C01778=1011.519,353.301,-157.245,170.736,52.593,160.409
C01779=1011.528,353.615,-157.291,170.746,52.587,160.410
C01780=1011.537,353.929,-157.337,170.758,52.582,160.411
C01781=1011.545,354.243,-157.384,170.769,52.577,160.412
C01782=1011.554,354.557,-157.431,170.779,52.571,160.412
C01783=1011.562,354.804,-157.467,170.788,52.567,160.413
C01784=1011.569,355.052,-157.505,170.796,52.563,160.414
C01785=1011.576,355.299,-157.541,170.806,52.558,160.414
C01786=1011.582,355.546,-157.578,170.814,52.554,160.415
C01787=1011.590,355.793,-157.615,170.823,52.550,160.416
C01788=1011.597,356.041,-157.652,170.831,52.546,160.416
C01789=1011.604,356.287,-157.689,170.840,52.541,160.417
C01790=1011.612,356.534,-157.726,170.849,52.537,160.418
C01791=1011.619,356.782,-157.762,170.859,52.533,160.419
C01792=1011.626,357.029,-157.800,170.867,52.529,160.420
C01793=1011.633,357.276,-157.836,170.876,52.525,160.420
C01794=1011.641,357.523,-157.873,170.884,52.521,160.421
C01795=1011.648,357.770,-157.911,170.893,52.517,160.422
C01796=1011.655,358.018,-157.948,170.903,52.513,160.423
C01797=1011.662,358.265,-157.985,170.911,52.509,160.423
C01798=1011.669,358.512,-158.023,170.920,52.505,160.424
C01799=1011.676,358.759,-158.060,170.928,52.500,160.425
C01800=1011.683,359.006,-158.097,170.937,52.497,160.425
C01801=1011.690,359.253,-158.135,170.947,52.492,160.426
C01802=1011.698,359.500,-158.172,170.956,52.489,160.427
C01803=1011.705,359.747,-158.210,170.964,52.485,160.428
C01804=1011.712,359.994,-158.248,170.973,52.481,160.428
C01805=1011.719,360.241,-158.285,170.983,52.477,160.429
C01806=1011.727,360.489,-158.323,170.991,52.473,160.430
C01807=1011.734,360.736,-158.360,171.000,52.469,160.431
C01808=1011.741,360.983,-158.398,171.009,52.465,160.432
C01809=1011.749,361.229,-158.436,171.019,52.461,160.433
C01810=1011.756,361.476,-158.473,171.027,52.457,160.433
C01811=1011.763,361.724,-158.511,171.036,52.453,160.434
C01812=1011.770,361.971,-158.548,171.045,52.450,160.435
C01813=1011.778,362.217,-158.587,171.055,52.445,160.436
C01814=1011.785,362.464,-158.624,171.064,52.442,160.437
C01815=1011.793,362.712,-158.662,171.073,52.438,160.438
C01816=1011.800,362.959,-158.700,171.082,52.434,160.438
C01817=1011.808,363.206,-158.738,171.091,52.430,160.439
C01818=1011.815,363.453,-158.775,171.100,52.427,160.440
C01819=1011.823,363.700,-158.814,171.110,52.423,160.441
C01820=1011.830,363.947,-158.851,171.119,52.419,160.442
C01821=1011.838,364.194,-158.890,171.128,52.415,160.443
C01822=1011.845,364.441,-158.927,171.138,52.411,160.444
C01823=1011.853,364.688,-158.966,171.147,52.408,160.445
C01824=1011.860,364.934,-159.004,171.156,52.404,160.446
C01825=1011.868,365.182,-159.042,171.166,52.400,160.447
C01826=1011.876,365.428,-159.080,171.175,52.397,160.447
C01827=1011.883,365.676,-159.117,171.184,52.392,160.448
C01828=1011.891,365.923,-159.156,171.193,52.389,160.449
C01829=1011.899,366.169,-159.194,171.202,52.385,160.450
C01830=1011.907,366.416,-159.233,171.212,52.382,160.451
C01831=1011.914,366.664,-159.270,171.221,52.378,160.452
C01832=1011.921,366.910,-159.309,171.232,52.375,160.453
C01833=1011.929,367.158,-159.348,171.241,52.371,160.454
C01834=1011.937,367.404,-159.386,171.250,52.368,160.455
C01835=1011.943,367.651,-159.425,171.260,52.364,160.456
C01836=1011.952,367.898,-159.464,171.269,52.360,160.457
C01837=1011.959,368.144,-159.503,171.279,52.356,160.458
C01838=1011.967,368.392,-159.542,171.288,52.354,160.459
C01839=1011.974,368.615,-159.577,171.297,52.350,160.460
C01840=1011.981,368.838,-159.612,171.305,52.347,160.461
C01841=1011.988,369.062,-159.646,171.314,52.343,160.461
C01842=1011.994,369.285,-159.682,171.322,52.341,160.462
C01843=1012.001,369.508,-159.716,171.331,52.337,160.463
C01844=1012.008,369.731,-159.752,171.339,52.334,160.464
C01845=1012.015,369.954,-159.787,171.349,52.332,160.465
C01846=1012.022,370.178,-159.822,171.358,52.328,160.466
C01847=1012.030,370.425,-159.861,171.367,52.325,160.467
C01848=1012.038,370.671,-159.900,171.377,52.321,160.468
C01849=1012.045,370.918,-159.939,171.386,52.318,160.469
C01850=1012.054,371.165,-159.978,171.396,52.314,160.470
C01851=1012.062,371.412,-160.017,171.406,52.312,160.471
C01852=1012.069,371.658,-160.057,171.416,52.308,160.472
C01853=1012.077,371.905,-160.095,171.425,52.305,160.473
C01854=1012.086,372.152,-160.134,171.435,52.301,160.474
C01855=1012.093,372.400,-160.174,171.445,52.298,160.476
C01856=1012.101,372.645,-160.213,171.455,52.295,160.477
C01857=1012.109,372.893,-160.251,171.465,52.291,160.478
C01858=1012.117,373.140,-160.291,171.474,52.288,160.479
C01859=1012.125,373.386,-160.330,171.485,52.285,160.480
C01860=1012.134,373.633,-160.370,171.494,52.281,160.481
C01861=1012.140,373.880,-160.409,171.504,52.278,160.482
C01862=1012.149,374.126,-160.448,171.514,52.275,160.483
C01863=1012.157,374.373,-160.487,171.524,52.272,160.484
C01864=1012.165,374.620,-160.527,171.534,52.269,160.486
C01865=1012.174,374.866,-160.567,171.545,52.265,160.487
C01866=1012.181,375.113,-160.606,171.554,52.262,160.488
C01867=1012.190,375.360,-160.646,171.564,52.259,160.489
C01868=1012.197,375.607,-160.686,171.575,52.256,160.490
C01869=1012.205,375.854,-160.726,171.584,52.253,160.491
C01870=1012.214,376.100,-160.765,171.595,52.250,160.493
C01871=1012.222,376.346,-160.806,171.604,52.247,160.494
C01872=1012.229,376.593,-160.845,171.614,52.244,160.495
C01873=1012.238,376.840,-160.885,171.625,52.240,160.496
C01874=1012.246,377.087,-160.925,171.635,52.237,160.497
C01875=1012.254,377.333,-160.965,171.645,52.234,160.498
C01876=1012.262,377.580,-161.005,171.656,52.232,160.500
C01877=1012.270,377.826,-161.045,171.666,52.228,160.501
C01878=1012.278,378.073,-161.085,171.675,52.225,160.502
C01879=1011.940,375.995,-161.099,171.571,52.309,160.503
C01880=1011.932,375.748,-161.059,171.561,52.312,160.502
C01881=1011.924,375.502,-161.019,171.551,52.315,160.501
C01882=1011.916,375.255,-160.980,171.541,52.318,160.500
C01883=1011.908,375.008,-160.940,171.531,52.322,160.499
C01884=1011.900,374.762,-160.900,171.521,52.324,160.497
C01885=1011.892,374.515,-160.860,171.511,52.328,160.496
C01886=1011.884,374.268,-160.822,171.500,52.331,160.495
C01887=1011.877,374.022,-160.782,171.491,52.335,160.494
C01888=1011.868,373.775,-160.743,171.481,52.338,160.493
C01889=1011.860,373.528,-160.704,171.472,52.341,160.492
C01890=1011.852,373.281,-160.664,171.461,52.344,160.491
C01891=1011.844,373.034,-160.625,171.451,52.348,160.490
C01892=1011.836,372.788,-160.587,171.442,52.351,160.489
C01893=1011.829,372.541,-160.547,171.431,52.354,160.487
C01894=1011.820,372.294,-160.508,171.422,52.358,160.486
C01895=1011.812,372.047,-160.469,171.412,52.361,160.485
C01896=1011.805,371.801,-160.429,171.402,52.364,160.484
C01897=1011.797,371.554,-160.391,171.393,52.368,160.483
C01898=1011.788,371.307,-160.351,171.382,52.371,160.482
C01899=1011.782,371.060,-160.313,171.373,52.374,160.481
C01900=1011.773,370.813,-160.274,171.363,52.378,160.480
C01901=1011.765,370.566,-160.235,171.354,52.381,160.479
C01902=1011.758,370.319,-160.196,171.344,52.384,160.478
C01903=1011.750,370.072,-160.157,171.334,52.388,160.477
C01904=1011.738,369.670,-160.093,171.318,52.394,160.475
C01905=1011.725,369.267,-160.030,171.302,52.400,160.473
C01906=1011.712,368.863,-159.967,171.287,52.405,160.472
C01907=1011.700,368.460,-159.904,171.272,52.411,160.470
C01908=1011.692,368.213,-159.865,171.261,52.414,160.469
C01909=1011.685,367.967,-159.827,171.252,52.418,160.468
C01910=1011.677,367.720,-159.787,171.243,52.422,160.467
C01911=1011.669,367.473,-159.749,171.234,52.425,160.466
C01912=1011.662,367.227,-159.711,171.224,52.429,160.465
C01913=1011.655,366.978,-159.672,171.214,52.432,160.464
C01914=1011.647,366.732,-159.634,171.204,52.436,160.463
C01915=1011.640,366.485,-159.596,171.195,52.439,160.462
C01916=1011.631,366.238,-159.557,171.186,52.443,160.461
C01917=1011.624,365.992,-159.519,171.176,52.447,160.460
C01918=1011.617,365.745,-159.481,171.167,52.450,160.459
C01919=1011.609,365.497,-159.443,171.157,52.454,160.458
C01920=1011.601,365.251,-159.404,171.148,52.458,160.458
C01921=1011.594,365.004,-159.367,171.139,52.461,160.457
C01922=1011.586,364.756,-159.328,171.130,52.466,160.456
C01923=1011.578,364.509,-159.291,171.121,52.469,160.455
C01924=1011.571,364.263,-159.252,171.111,52.473,160.454
C01925=1011.564,364.016,-159.215,171.102,52.477,160.453
C01926=1011.556,363.769,-159.177,171.093,52.480,160.452
C01927=1011.549,363.521,-159.138,171.083,52.484,160.451
C01928=1011.542,363.274,-159.101,171.074,52.488,160.451
C01929=1011.534,363.027,-159.062,171.065,52.492,160.450
C01930=1011.527,362.780,-159.025,171.055,52.496,160.449
C01931=1011.520,362.533,-158.987,171.047,52.500,160.448
C01932=1011.512,362.287,-158.949,171.038,52.503,160.447
C01933=1011.505,362.039,-158.912,171.028,52.507,160.446
C01934=1011.498,361.792,-158.874,171.019,52.511,160.445
C01935=1011.490,361.545,-158.837,171.010,52.515,160.445
C01936=1011.483,361.299,-158.798,171.001,52.519,160.444
C01937=1011.476,361.052,-158.761,170.992,52.523,160.443
C01938=1011.468,360.804,-158.723,170.983,52.526,160.442
C01939=1011.461,360.557,-158.686,170.974,52.531,160.441
C01940=1011.454,360.310,-158.648,170.964,52.534,160.440
C01941=1011.447,360.063,-158.611,170.956,52.539,160.440
C01942=1011.439,359.816,-158.573,170.947,52.543,160.439
C01943=1011.432,359.569,-158.536,170.937,52.547,160.438
C01944=1011.425,359.322,-158.498,170.929,52.551,160.437
C01945=1011.418,359.074,-158.461,170.920,52.554,160.436
C01946=1011.410,358.827,-158.423,170.911,52.558,160.436
C01947=1011.403,358.580,-158.386,170.903,52.563,160.435
C01948=1011.396,358.333,-158.348,170.893,52.567,160.434
C01949=1011.390,358.086,-158.312,170.884,52.571,160.433
C01950=1011.382,357.839,-158.275,170.876,52.575,160.433
C01951=1011.374,357.592,-158.237,170.867,52.579,160.432
C01952=1011.367,357.344,-158.200,170.857,52.583,160.431
C01953=1011.360,357.097,-158.163,170.849,52.587,160.430
C01954=1011.353,356.851,-158.126,170.840,52.591,160.430
C01955=1011.346,356.603,-158.089,170.831,52.595,160.429
C01956=1011.339,356.356,-158.052,170.823,52.600,160.428
C01957=1011.332,356.108,-158.015,170.813,52.604,160.427
C01958=1011.324,355.862,-157.978,170.805,52.608,160.427
C01959=1011.317,355.614,-157.942,170.796,52.612,160.426
C01960=1011.310,355.367,-157.905,170.787,52.616,160.425
C01961=1011.303,355.121,-157.868,170.779,52.620,160.424
C01962=1011.296,354.873,-157.831,170.770,52.624,160.424
C01963=1011.289,354.625,-157.795,170.761,52.629,160.423
C01964=1011.280,354.309,-157.748,170.751,52.634,160.422
C01965=1011.271,353.993,-157.701,170.739,52.640,160.421
C01966=1011.262,353.677,-157.654,170.728,52.646,160.421
C01967=1011.253,353.361,-157.607,170.717,52.651,160.420
C01968=1011.246,353.113,-157.570,170.708,52.655,160.419
C01969=1011.240,352.866,-157.534,170.699,52.659,160.418
C01970=1011.232,352.619,-157.498,170.691,52.664,160.418
C01971=1011.226,352.372,-157.461,170.683,52.668,160.417
C01972=1011.218,352.124,-157.425,170.674,52.673,160.416
C01973=1011.212,351.877,-157.389,170.666,52.677,160.416
C01974=1011.204,351.630,-157.352,170.657,52.681,160.415
C01975=1011.198,351.383,-157.316,170.649,52.686,160.415
C01976=1011.190,351.135,-157.280,170.639,52.690,160.414
C01977=1011.184,350.888,-157.243,170.631,52.695,160.413
C01978=1011.176,350.641,-157.207,170.623,52.699,160.413
C01979=1011.170,350.393,-157.171,170.614,52.703,160.412
C01980=1011.163,350.146,-157.136,170.606,52.708,160.411
C01981=1011.156,349.899,-157.099,170.597,52.712,160.411
C01982=1011.149,349.652,-157.063,170.589,52.717,160.410
C01983=1011.142,349.404,-157.026,170.581,52.721,160.410
C01984=1011.135,349.157,-156.991,170.573,52.726,160.409
C01985=1011.129,348.910,-156.954,170.564,52.730,160.408
C01986=1011.122,348.663,-156.919,170.556,52.735,160.408
C01987=1011.115,348.415,-156.883,170.548,52.739,160.407
C01988=1011.108,348.168,-156.847,170.539,52.744,160.407
C01989=1011.102,347.920,-156.811,170.531,52.749,160.406
C01990=1011.095,347.673,-156.775,170.523,52.753,160.406
C01991=1011.088,347.425,-156.739,170.515,52.758,160.405
C01992=1011.081,347.178,-156.703,170.505,52.762,160.404
C01993=1011.075,346.931,-156.667,170.497,52.767,160.404
C01994=1011.068,346.684,-156.632,170.489,52.772,160.403
C01995=1011.062,346.436,-156.596,170.480,52.776,160.403
C01996=1011.055,346.189,-156.560,170.472,52.781,160.402
C01997=1011.048,345.941,-156.525,170.464,52.786,160.402
C01998=1011.042,345.694,-156.489,170.456,52.791,160.401
C01999=1011.035,345.446,-156.454,170.447,52.795,160.401
C02000=1011.028,345.200,-156.418,170.439,52.800,160.400
C02001=1011.022,344.952,-156.382,170.431,52.805,160.400
C02002=1011.015,344.705,-156.347,170.423,52.809,160.399
C02003=1011.008,344.457,-156.312,170.415,52.814,160.399
C02004=1011.002,344.210,-156.277,170.407,52.819,160.398
C02005=1010.995,343.962,-156.242,170.399,52.824,160.398
C02006=1010.989,343.715,-156.206,170.391,52.829,160.397
C02007=1010.982,343.467,-156.171,170.383,52.834,160.397
C02008=1010.975,343.220,-156.136,170.375,52.838,160.396
C02009=1010.968,342.973,-156.100,170.366,52.843,160.396
C02010=1010.962,342.725,-156.065,170.358,52.848,160.395
C02011=1010.956,342.478,-156.030,170.350,52.853,160.395
C02012=1010.949,342.230,-155.994,170.343,52.857,160.395
C02013=1010.942,341.983,-155.959,170.335,52.862,160.394
C02014=1010.936,341.735,-155.924,170.327,52.867,160.394
C02015=1010.929,341.488,-155.888,170.319,52.872,160.393
C02016=1010.923,341.241,-155.853,170.311,52.877,160.393
C02017=1010.916,340.993,-155.819,170.303,52.881,160.392
C02018=1010.909,340.745,-155.784,170.294,52.886,160.392
C02019=1010.903,340.498,-155.749,170.286,52.891,160.391
C02020=1010.897,340.251,-155.713,170.279,52.897,160.391
C02021=1010.891,340.003,-155.679,170.271,52.901,160.390
C02022=1010.884,339.755,-155.644,170.263,52.906,160.390
C02023=1010.877,339.508,-155.609,170.254,52.911,160.390
C02024=1010.869,339.189,-155.564,170.245,52.917,160.389
C02025=1010.861,338.871,-155.519,170.234,52.924,160.388
C02026=1010.853,338.551,-155.474,170.224,52.930,160.388
C02027=1010.844,338.233,-155.429,170.214,52.937,160.387
C02028=1010.838,337.985,-155.395,170.206,52.943,160.387
C02029=1010.832,337.738,-155.360,170.198,52.947,160.387
C02030=1010.825,337.490,-155.326,170.191,52.952,160.386
C02031=1010.819,337.242,-155.291,170.183,52.957,160.386
C02032=1010.813,336.996,-155.257,170.175,52.962,160.386
C02033=1010.806,336.748,-155.222,170.168,52.968,160.385
C02034=1010.800,336.500,-155.188,170.159,52.973,160.385
C02035=1010.794,336.252,-155.154,170.152,52.978,160.385
C02036=1010.787,336.005,-155.119,170.144,52.983,160.384
C02037=1010.780,335.757,-155.085,170.136,52.988,160.384
C02038=1010.774,335.510,-155.051,170.128,52.993,160.383
C02039=1010.768,335.262,-155.016,170.120,52.999,160.383
C02040=1010.762,335.015,-154.982,170.113,53.003,160.383
C02041=1010.755,334.767,-154.948,170.105,53.009,160.382
C02042=1010.749,334.519,-154.914,170.098,53.014,160.382
C02043=1010.743,334.271,-154.879,170.090,53.019,160.382
C02044=1010.737,334.024,-154.845,170.082,53.025,160.381
C02045=1010.731,333.776,-154.811,170.074,53.030,160.381
C02046=1010.725,333.529,-154.777,170.066,53.035,160.381
C02047=1010.718,333.281,-154.743,170.059,53.040,160.380
C02048=1010.712,333.034,-154.709,170.052,53.046,160.380
C02049=1010.705,332.786,-154.674,170.044,53.050,160.380
C02050=1010.699,332.539,-154.640,170.036,53.056,160.380
C02051=1010.693,332.291,-154.606,170.029,53.061,160.379
C02052=1010.687,332.043,-154.572,170.021,53.067,160.379
C02053=1010.681,331.796,-154.538,170.013,53.072,160.379
C02054=1010.675,331.548,-154.503,170.006,53.077,160.378
C02055=1010.668,331.301,-154.471,169.999,53.082,160.378
C02056=1010.663,331.053,-154.437,169.991,53.088,160.378
C02057=1010.656,330.805,-154.402,169.983,53.093,160.378
C02058=1010.650,330.558,-154.370,169.976,53.099,160.377
C02059=1010.643,330.310,-154.335,169.968,53.104,160.377
C02060=1010.637,330.062,-154.301,169.960,53.110,160.377
C02061=1010.631,329.815,-154.268,169.954,53.115,160.377
C02062=1010.625,329.568,-154.234,169.946,53.121,160.376
C02063=1010.618,329.319,-154.201,169.938,53.126,160.376
C02064=1010.613,329.072,-154.167,169.931,53.132,160.376
C02065=1010.607,328.824,-154.134,169.923,53.137,160.376
C02066=1010.600,328.577,-154.100,169.915,53.143,160.375
C02067=1010.594,328.328,-154.067,169.909,53.148,160.375
C02068=1010.589,328.081,-154.033,169.901,53.153,160.375
C02069=1010.582,327.834,-154.000,169.893,53.159,160.375
C02070=1010.577,327.586,-153.966,169.886,53.164,160.374
C02071=1010.571,327.338,-153.932,169.878,53.170,160.374
C02072=1010.564,327.090,-153.899,169.871,53.175,160.374
C02073=1010.558,326.842,-153.866,169.864,53.181,160.374
C02074=1010.552,326.595,-153.833,169.857,53.187,160.374
C02075=1010.546,326.347,-153.799,169.849,53.192,160.373
C02076=1010.541,326.099,-153.766,169.841,53.198,160.373
C02077=1010.534,325.852,-153.733,169.835,53.203,160.373
C02078=1010.528,325.605,-153.699,169.827,53.209,160.373
C02079=1010.523,325.357,-153.666,169.820,53.215,160.373
C02080=1010.517,325.109,-153.633,169.812,53.220,160.372
C02081=1010.510,324.861,-153.600,169.804,53.226,160.372
C02082=1010.504,324.614,-153.567,169.798,53.232,160.372
C02083=1010.498,324.366,-153.535,169.791,53.237,160.372
C02084=1010.490,324.042,-153.492,169.780,53.245,160.371
C02085=1010.482,323.719,-153.449,169.772,53.252,160.371
C02086=1010.474,323.396,-153.407,169.761,53.260,160.371
C02087=1010.467,323.073,-153.364,169.753,53.267,160.371
C02088=1010.460,322.825,-153.331,169.745,53.273,160.371
C02089=1010.454,322.577,-153.299,169.738,53.279,160.371
C02090=1010.448,322.330,-153.266,169.730,53.285,160.370
C02091=1010.442,322.082,-153.234,169.723,53.291,160.370
C02092=1010.436,321.834,-153.200,169.716,53.296,160.370
C02093=1010.430,321.586,-153.168,169.709,53.302,160.370
C02094=1010.423,321.339,-153.135,169.702,53.308,160.370
C02095=1010.418,321.090,-153.103,169.694,53.314,160.370
C02096=1010.411,320.843,-153.070,169.688,53.320,160.370
C02097=1010.406,320.594,-153.038,169.681,53.325,160.370
C02098=1010.400,320.347,-153.005,169.673,53.331,160.369
C02099=1010.394,320.100,-152.972,169.666,53.337,160.369
C02100=1010.388,319.852,-152.940,169.659,53.343,160.369
C02101=1010.382,319.604,-152.908,169.652,53.349,160.369
C02102=1010.376,319.356,-152.876,169.645,53.355,160.369
C02103=1010.371,319.109,-152.843,169.638,53.361,160.369
C02104=1010.365,318.860,-152.811,169.630,53.367,160.369
C02105=1010.358,318.613,-152.778,169.624,53.372,160.369
C02106=1010.352,318.364,-152.746,169.617,53.378,160.369
C02107=1010.347,318.117,-152.714,169.609,53.385,160.369
C02108=1010.341,317.869,-152.681,169.602,53.391,160.368
C02109=1010.336,317.621,-152.649,169.595,53.396,160.368
C02110=1010.330,317.374,-152.616,169.588,53.402,160.368
C02111=1010.324,317.126,-152.584,169.581,53.408,160.368
C02112=1010.318,316.878,-152.552,169.574,53.415,160.368
C02113=1010.312,316.631,-152.520,169.567,53.420,160.368
C02114=1010.307,316.382,-152.487,169.560,53.426,160.368
C02115=1010.301,316.134,-152.455,169.553,53.432,160.368
C02116=1010.296,315.886,-152.424,169.546,53.439,160.368
C02117=1010.289,315.639,-152.391,169.540,53.444,160.368
C02118=1010.284,315.391,-152.359,169.532,53.451,160.368
C02119=1010.278,315.143,-152.327,169.525,53.457,160.368
C02120=1010.273,314.895,-152.295,169.518,53.463,160.368
C02121=1010.267,314.647,-152.263,169.511,53.468,160.367
C02122=1010.262,314.400,-152.231,169.504,53.474,160.367
C02123=1010.256,314.152,-152.199,169.497,53.481,160.367
C02124=1010.250,313.904,-152.167,169.490,53.487,160.367
C02125=1010.244,313.656,-152.135,169.484,53.493,160.367
C02126=1010.240,313.408,-152.103,169.476,53.499,160.367
C02127=1010.234,313.160,-152.071,169.469,53.505,160.367
C02128=1010.228,312.913,-152.039,169.463,53.511,160.367
C02129=1010.222,312.664,-152.007,169.456,53.517,160.367
C02130=1010.217,312.417,-151.975,169.449,53.524,160.367
C02131=1010.211,312.169,-151.943,169.443,53.529,160.367
C02132=1010.206,311.921,-151.911,169.436,53.536,160.367
C02133=1010.201,311.673,-151.879,169.429,53.543,160.367
C02134=1010.195,311.425,-151.847,169.421,53.549,160.367
C02135=1010.189,311.178,-151.816,169.415,53.555,160.367
C02136=1010.184,310.930,-151.784,169.408,53.561,160.367
C02137=1010.178,310.682,-151.752,169.401,53.567,160.367
C02138=1010.173,310.434,-151.721,169.395,53.573,160.367
C02139=1010.168,310.186,-151.689,169.388,53.579,160.367
C02140=1010.162,309.938,-151.657,169.381,53.586,160.367
C02141=1010.157,309.690,-151.625,169.375,53.592,160.367
C02142=1010.152,309.443,-151.593,169.368,53.598,160.367
C02143=1010.146,309.195,-151.562,169.360,53.605,160.367
C02144=1010.140,308.877,-151.521,169.352,53.613,160.367
C02145=1010.133,308.560,-151.481,169.343,53.621,160.367
C02146=1010.126,308.242,-151.440,169.335,53.629,160.367
C02147=1010.118,307.925,-151.401,169.326,53.637,160.367
C02148=1010.112,307.676,-151.371,169.320,53.644,160.367
C02149=1010.106,307.429,-151.339,169.313,53.650,160.367
C02150=1010.101,307.181,-151.309,169.306,53.657,160.368
C02151=1010.096,306.933,-151.278,169.300,53.663,160.368
C02152=1010.090,306.685,-151.246,169.292,53.669,160.368
C02153=1010.084,306.437,-151.215,169.286,53.676,160.368
C02154=1010.079,306.188,-151.184,169.279,53.682,160.368
C02155=1010.073,305.941,-151.154,169.273,53.689,160.368
C02156=1010.068,305.692,-151.123,169.266,53.695,160.368
C02157=1010.062,305.445,-151.092,169.259,53.702,160.368
C02158=1010.056,305.196,-151.061,169.252,53.708,160.368
C02159=1010.050,304.949,-151.030,169.246,53.715,160.368
C02160=1010.045,304.700,-150.999,169.240,53.722,160.368
C02161=1010.039,304.453,-150.969,169.232,53.728,160.368
C02162=1010.034,304.204,-150.938,169.227,53.735,160.369
C02163=1010.028,303.957,-150.908,169.219,53.741,160.368
C02164=1010.023,303.709,-150.877,169.213,53.748,160.369
C02165=1010.017,303.461,-150.846,169.206,53.754,160.368
C02166=1010.012,303.213,-150.815,169.200,53.761,160.369
C02167=1010.007,302.965,-150.785,169.193,53.768,160.369
C02168=1010.002,302.717,-150.754,169.186,53.774,160.369
C02169=1009.996,302.469,-150.724,169.180,53.781,160.369
C02170=1009.991,302.221,-150.693,169.174,53.788,160.369
C02171=1009.985,301.973,-150.663,169.166,53.794,160.369
C02172=1009.980,301.725,-150.632,169.160,53.801,160.369
C02173=1009.974,301.477,-150.601,169.154,53.807,160.370
C02174=1009.969,301.229,-150.570,169.147,53.814,160.370
C02175=1009.963,300.981,-150.540,169.140,53.821,160.370
C02176=1009.958,300.733,-150.509,169.135,53.827,160.370
C02177=1009.952,300.484,-150.479,169.128,53.834,160.370
C02178=1009.947,300.236,-150.448,169.121,53.841,160.370
C02179=1009.942,299.988,-150.418,169.114,53.848,160.370
C02180=1009.936,299.740,-150.387,169.108,53.854,160.370
C02181=1009.931,299.492,-150.357,169.102,53.861,160.371
C02182=1009.926,299.244,-150.327,169.095,53.868,160.371
C02183=1009.921,298.997,-150.297,169.089,53.875,160.371
C02184=1009.916,298.748,-150.266,169.082,53.881,160.371
C02185=1009.910,298.500,-150.236,169.075,53.888,160.371
C02186=1009.905,298.252,-150.205,169.070,53.894,160.371
C02187=1009.899,298.004,-150.175,169.063,53.901,160.371
C02188=1009.894,297.755,-150.144,169.056,53.908,160.372
C02189=1009.889,297.508,-150.114,169.051,53.915,160.372
C02190=1009.884,297.260,-150.083,169.044,53.922,160.372
C02191=1009.879,297.012,-150.054,169.037,53.929,160.372
C02192=1009.873,296.763,-150.023,169.031,53.936,160.372
C02193=1009.869,296.516,-149.994,169.025,53.943,160.373
C02194=1009.863,296.268,-149.963,169.018,53.950,160.373
C02195=1009.858,296.019,-149.933,169.012,53.957,160.373
C02196=1009.853,295.771,-149.902,169.006,53.963,160.373
C02197=1009.849,295.523,-149.872,168.999,53.970,160.373
C02198=1009.843,295.275,-149.842,168.993,53.977,160.373
C02199=1009.838,295.026,-149.812,168.987,53.984,160.374
C02200=1009.831,294.680,-149.770,168.978,53.993,160.374
C02201=1009.824,294.334,-149.728,168.969,54.003,160.374
C02202=1009.816,293.987,-149.685,168.960,54.013,160.374
C02203=1009.809,293.641,-149.644,168.951,54.022,160.375
C02204=1009.570,294.619,-150.127,168.951,54.055,160.382
C02205=1009.577,294.883,-150.159,168.958,54.048,160.382
C02206=1009.581,295.148,-150.191,168.964,54.041,160.382
C02207=1009.586,295.412,-150.224,168.971,54.034,160.382
C02208=1009.592,295.678,-150.256,168.978,54.026,160.381
C02209=1009.598,295.926,-150.286,168.984,54.019,160.381
C02210=1009.602,296.174,-150.316,168.991,54.012,160.381
C02211=1009.608,296.422,-150.346,168.997,54.005,160.381
C02212=1009.612,296.670,-150.377,169.003,53.998,160.381
C02213=1009.618,296.918,-150.407,169.010,53.992,160.381
C02214=1009.622,297.166,-150.437,169.017,53.985,160.381
C02215=1009.628,297.414,-150.467,169.022,53.979,160.380
C02216=1009.633,297.663,-150.497,169.029,53.972,160.380
C02217=1009.638,297.910,-150.527,169.036,53.965,160.380
C02218=1009.643,298.158,-150.558,169.041,53.958,160.380
C02219=1009.649,298.407,-150.588,169.048,53.951,160.380
C02220=1009.654,298.655,-150.619,169.055,53.944,160.379
C02221=1009.659,298.903,-150.648,169.062,53.938,160.380
C02222=1009.664,299.151,-150.679,169.068,53.931,160.379
C02223=1009.670,299.398,-150.709,169.074,53.924,160.379
C02224=1009.674,299.647,-150.740,169.081,53.917,160.379
C02225=1009.680,299.895,-150.770,169.087,53.910,160.379
C02226=1009.685,300.143,-150.801,169.094,53.904,160.379
C02227=1009.691,300.391,-150.831,169.101,53.897,160.379
C02228=1009.696,300.640,-150.862,169.107,53.890,160.379
C02229=1009.703,300.980,-150.904,169.115,53.882,160.378
C02230=1009.711,301.321,-150.945,169.124,53.872,160.378
C02231=1009.717,301.662,-150.988,169.133,53.863,160.378
C02232=1009.725,302.004,-151.029,169.142,53.854,160.378
C02233=1009.731,302.252,-151.060,169.149,53.848,160.378
C02234=1009.736,302.500,-151.091,169.156,53.841,160.378
C02235=1009.742,302.748,-151.121,169.163,53.834,160.378
C02236=1009.747,302.996,-151.152,169.169,53.828,160.378
C02237=1009.753,303.244,-151.182,169.176,53.821,160.377
C02238=1009.758,303.492,-151.213,169.183,53.814,160.377
C02239=1009.764,303.740,-151.244,169.190,53.807,160.377
C02240=1009.769,303.988,-151.275,169.195,53.801,160.377
C02241=1009.774,304.236,-151.305,169.202,53.795,160.377
C02242=1009.780,304.484,-151.336,169.209,53.788,160.377
C02243=1009.785,304.731,-151.366,169.215,53.782,160.377
C02244=1009.790,304.980,-151.397,169.222,53.775,160.377
C02245=1009.796,305.227,-151.427,169.229,53.769,160.377
C02246=1009.801,305.476,-151.458,169.236,53.762,160.377
C02247=1009.807,305.723,-151.489,169.242,53.756,160.377
C02248=1009.813,305.972,-151.521,169.249,53.749,160.377
C02249=1009.819,306.219,-151.551,169.256,53.742,160.377
C02250=1009.824,306.468,-151.582,169.262,53.736,160.376
C02251=1009.830,306.715,-151.612,169.269,53.730,160.376
C02252=1009.835,306.964,-151.643,169.275,53.723,160.376
C02253=1009.841,307.211,-151.674,169.283,53.716,160.376
C02254=1009.847,307.460,-151.706,169.290,53.710,160.376
C02255=1009.852,307.708,-151.737,169.296,53.703,160.376
C02256=1009.858,307.956,-151.767,169.303,53.697,160.376
C02257=1009.866,308.275,-151.808,169.312,53.688,160.376
C02258=1009.872,308.595,-151.848,169.321,53.681,160.376
C02259=1009.879,308.915,-151.888,169.329,53.672,160.376
C02260=1009.886,309.235,-151.929,169.337,53.665,160.376
C02261=1009.892,309.482,-151.961,169.345,53.658,160.376
C02262=1009.896,309.731,-151.992,169.351,53.651,160.376
C02263=1009.902,309.979,-152.024,169.358,53.646,160.376
C02264=1009.907,310.226,-152.056,169.365,53.639,160.376
C02265=1009.913,310.474,-152.088,169.372,53.633,160.376
C02266=1009.918,310.722,-152.118,169.378,53.627,160.376
C02267=1009.924,310.970,-152.150,169.385,53.621,160.376
C02268=1009.929,311.218,-152.183,169.392,53.615,160.376
C02269=1009.934,311.466,-152.214,169.399,53.608,160.376
C02270=1009.940,311.714,-152.246,169.405,53.602,160.376
C02271=1009.945,311.961,-152.278,169.412,53.596,160.376
C02272=1009.951,312.209,-152.310,169.420,53.589,160.376
C02273=1009.957,312.457,-152.342,169.426,53.583,160.376
C02274=1009.961,312.705,-152.374,169.433,53.577,160.376
C02275=1009.967,312.952,-152.406,169.440,53.571,160.376
C02276=1009.973,313.201,-152.438,169.447,53.565,160.376
C02277=1009.978,313.448,-152.469,169.453,53.559,160.376
C02278=1009.984,313.696,-152.501,169.461,53.553,160.376
C02279=1009.989,313.944,-152.533,169.468,53.546,160.376
C02280=1009.995,314.192,-152.566,169.474,53.540,160.376
C02281=1010.000,314.440,-152.597,169.481,53.534,160.376
C02282=1010.005,314.687,-152.629,169.488,53.528,160.377
C02283=1010.011,314.936,-152.661,169.496,53.522,160.377
C02284=1010.017,315.184,-152.693,169.502,53.517,160.377
C02285=1010.023,315.431,-152.725,169.509,53.510,160.377
C02286=1010.028,315.679,-152.758,169.517,53.504,160.377
C02287=1010.034,315.927,-152.790,169.524,53.498,160.377
C02288=1010.040,316.175,-152.822,169.530,53.492,160.377
C02289=1010.045,316.422,-152.853,169.537,53.486,160.377
C02290=1010.051,316.671,-152.885,169.545,53.480,160.377
C02291=1010.057,316.917,-152.918,169.552,53.474,160.377
C02292=1010.062,317.166,-152.950,169.558,53.468,160.377
C02293=1010.068,317.414,-152.982,169.565,53.462,160.377
C02294=1010.074,317.661,-153.015,169.572,53.456,160.377
C02295=1010.080,317.909,-153.047,169.580,53.450,160.378
C02296=1010.086,318.158,-153.079,169.587,53.444,160.378
C02297=1010.091,318.404,-153.111,169.593,53.438,160.378
C02298=1010.097,318.653,-153.144,169.601,53.432,160.378
C02299=1010.103,318.901,-153.176,169.608,53.426,160.378
C02300=1010.109,319.149,-153.209,169.615,53.420,160.378
C02301=1010.114,319.396,-153.240,169.622,53.415,160.378
C02302=1010.121,319.644,-153.273,169.629,53.409,160.378
C02303=1010.127,319.892,-153.305,169.636,53.402,160.378
C02304=1010.132,320.140,-153.338,169.644,53.397,160.379
C02305=1010.138,320.388,-153.370,169.651,53.391,160.379
C02306=1010.144,320.635,-153.403,169.658,53.385,160.379
C02307=1010.150,320.883,-153.435,169.665,53.379,160.379
C02308=1010.156,321.131,-153.468,169.672,53.373,160.379
C02309=1010.162,321.379,-153.501,169.680,53.367,160.379
C02310=1010.168,321.627,-153.533,169.687,53.361,160.379
C02311=1010.173,321.874,-153.565,169.694,53.356,160.380
C02312=1010.180,322.122,-153.598,169.701,53.350,160.380
C02313=1010.186,322.370,-153.630,169.709,53.344,160.380
C02314=1010.192,322.617,-153.663,169.716,53.338,160.380
C02315=1010.197,322.865,-153.696,169.723,53.332,160.380
C02316=1010.203,323.113,-153.728,169.731,53.326,160.380
C02317=1010.212,323.439,-153.771,169.740,53.319,160.381
C02318=1010.220,323.765,-153.815,169.750,53.311,160.381
C02319=1010.228,324.090,-153.857,169.759,53.304,160.381
C02320=1010.235,324.416,-153.900,169.769,53.297,160.381
C02321=1010.242,324.663,-153.933,169.776,53.291,160.381
C02322=1010.248,324.911,-153.966,169.784,53.285,160.382
C02323=1010.254,325.158,-153.999,169.791,53.279,160.382
C02324=1010.260,325.406,-154.032,169.798,53.274,160.382
C02325=1010.266,325.654,-154.065,169.805,53.268,160.382
C02326=1010.272,325.902,-154.098,169.813,53.263,160.382
C02327=1010.278,326.149,-154.131,169.821,53.257,160.383
C02328=1010.284,326.397,-154.165,169.828,53.251,160.383
C02329=1010.289,326.644,-154.198,169.834,53.246,160.383
C02330=1010.296,326.892,-154.231,169.842,53.240,160.383
C02331=1010.301,327.140,-154.264,169.850,53.235,160.384
C02332=1010.308,327.388,-154.299,169.857,53.229,160.384
C02333=1010.314,327.636,-154.331,169.865,53.224,160.384
C02334=1010.319,327.883,-154.365,169.873,53.218,160.384
C02335=1010.325,328.131,-154.399,169.879,53.213,160.385
C02336=1010.332,328.378,-154.432,169.887,53.207,160.385
C02337=1010.337,328.626,-154.466,169.895,53.202,160.385
C02338=1010.344,328.874,-154.499,169.902,53.196,160.385
C02339=1010.350,329.122,-154.532,169.910,53.191,160.386
C02340=1010.356,329.369,-154.566,169.918,53.185,160.386
C02341=1010.362,329.617,-154.599,169.924,53.180,160.386
C02342=1010.369,329.865,-154.633,169.932,53.174,160.386
C02343=1010.374,330.113,-154.667,169.940,53.169,160.387
C02344=1010.381,330.360,-154.700,169.947,53.163,160.387
C02345=1010.386,330.607,-154.733,169.955,53.158,160.387
C02346=1010.393,330.855,-154.768,169.962,53.152,160.387
C02347=1010.399,331.102,-154.801,169.970,53.147,160.388
C02348=1010.405,331.350,-154.835,169.977,53.142,160.388
C02349=1010.411,331.598,-154.869,169.984,53.136,160.388
C02350=1010.418,331.845,-154.903,169.993,53.131,160.389
C02351=1010.424,332.093,-154.937,170.000,53.126,160.389
C02352=1010.430,332.341,-154.970,170.008,53.120,160.389
C02353=1010.436,332.588,-155.004,170.015,53.115,160.389
C02354=1010.442,332.836,-155.039,170.024,53.110,160.390
C02355=1010.448,333.084,-155.073,170.030,53.105,160.390
C02356=1010.454,333.331,-155.107,170.038,53.099,160.390
C02357=1010.460,333.579,-155.141,170.046,53.094,160.391
C02358=1010.466,333.826,-155.175,170.054,53.089,160.391
C02359=1010.474,334.074,-155.209,170.061,53.083,160.391
C02360=1010.479,334.321,-155.243,170.069,53.078,160.392
C02361=1010.486,334.569,-155.278,170.077,53.073,160.392
C02362=1010.492,334.816,-155.312,170.085,53.067,160.392
C02363=1010.498,335.064,-155.346,170.093,53.063,160.393
C02364=1010.504,335.312,-155.380,170.099,53.058,160.393
C02365=1010.510,335.560,-155.415,170.108,53.053,160.394
C02366=1010.516,335.807,-155.449,170.115,53.047,160.394
C02367=1010.523,336.055,-155.483,170.123,53.042,160.394
C02368=1010.530,336.302,-155.518,170.131,53.037,160.395
C02369=1010.536,336.549,-155.552,170.139,53.031,160.395
C02370=1010.543,336.797,-155.586,170.147,53.026,160.395
C02371=1010.549,337.045,-155.620,170.155,53.022,160.396
C02372=1010.555,337.293,-155.655,170.162,53.016,160.396
C02373=1010.562,337.540,-155.690,170.171,53.011,160.397
C02374=1010.568,337.787,-155.724,170.178,53.006,160.397
C02375=1010.574,338.035,-155.758,170.186,53.001,160.397
C02376=1010.581,338.283,-155.793,170.194,52.996,160.398
C02377=1010.589,338.604,-155.838,170.204,52.990,160.398
C02378=1010.597,338.925,-155.883,170.215,52.983,160.399
C02379=1010.605,339.246,-155.929,170.224,52.977,160.399
C02380=1010.613,339.567,-155.974,170.235,52.970,160.400
C02381=1010.620,339.815,-156.009,170.243,52.965,160.400
C02382=1010.627,340.063,-156.043,170.251,52.960,160.401
C02383=1010.633,340.309,-156.078,170.259,52.955,160.401
C02384=1010.639,340.557,-156.113,170.267,52.950,160.402
C02385=1010.646,340.805,-156.148,170.275,52.945,160.402
C02386=1010.652,341.052,-156.183,170.283,52.940,160.403
C02387=1010.659,341.300,-156.219,170.291,52.935,160.403
C02388=1010.665,341.546,-156.253,170.299,52.930,160.403
C02389=1010.671,341.794,-156.288,170.306,52.926,160.404
C02390=1010.678,342.042,-156.323,170.314,52.921,160.404
C02391=1010.684,342.289,-156.359,170.322,52.916,160.405
C02392=1010.691,342.537,-156.394,170.330,52.911,160.405
C02393=1010.698,342.784,-156.429,170.338,52.906,160.406
C02394=1010.704,343.031,-156.464,170.347,52.901,160.406
C02395=1010.710,343.279,-156.500,170.355,52.896,160.407
C02396=1010.717,343.526,-156.535,170.363,52.892,160.407
C02397=1010.724,343.774,-156.570,170.371,52.887,160.407
C02398=1010.731,344.021,-156.605,170.379,52.882,160.408
C02399=1010.737,344.269,-156.641,170.387,52.877,160.408
C02400=1010.744,344.516,-156.676,170.395,52.872,160.409
C02401=1010.750,344.764,-156.711,170.404,52.868,160.410
C02402=1010.757,345.011,-156.746,170.412,52.863,160.410
C02403=1010.764,345.258,-156.781,170.421,52.858,160.411
C02404=1010.770,345.506,-156.817,170.429,52.853,160.411
C02405=1010.777,345.753,-156.853,170.437,52.848,160.412
C02406=1010.784,346.000,-156.888,170.446,52.844,160.412
C02407=1010.790,346.248,-156.924,170.454,52.839,160.413
C02408=1010.797,346.496,-156.959,170.462,52.835,160.413
C02409=1010.803,346.743,-156.996,170.470,52.830,160.414
C02410=1010.810,346.990,-157.031,170.479,52.826,160.414
C02411=1010.817,347.237,-157.067,170.487,52.821,160.415
C02412=1010.823,347.485,-157.103,170.495,52.816,160.415
C02413=1010.830,347.732,-157.139,170.503,52.812,160.416
C02414=1010.837,347.980,-157.174,170.511,52.807,160.417
C02415=1010.843,348.227,-157.211,170.520,52.803,160.417
C02416=1010.850,348.474,-157.246,170.528,52.798,160.418
C02417=1010.857,348.721,-157.282,170.537,52.794,160.418
C02418=1010.864,348.969,-157.318,170.545,52.789,160.419
C02419=1010.871,349.216,-157.354,170.553,52.785,160.420
C02420=1010.877,349.463,-157.390,170.561,52.780,160.420
C02421=1010.885,349.711,-157.426,170.570,52.776,160.421
C02422=1010.891,349.958,-157.462,170.579,52.770,160.421
C02423=1010.898,350.205,-157.498,170.588,52.766,160.422
C02424=1010.905,350.453,-157.535,170.596,52.761,160.423
C02425=1010.912,350.700,-157.570,170.604,52.757,160.423
C02426=1010.918,350.947,-157.606,170.613,52.753,160.424
C02427=1010.926,351.195,-157.643,170.621,52.748,160.424
C02428=1010.932,351.442,-157.679,170.629,52.744,160.425
C02429=1010.940,351.689,-157.715,170.638,52.740,160.426
C02430=1010.946,351.936,-157.752,170.646,52.735,160.426
C02431=1010.954,352.184,-157.788,170.656,52.731,160.427
C02432=1010.960,352.431,-157.824,170.664,52.726,160.428
C02433=1010.967,352.677,-157.860,170.673,52.722,160.428
C02434=1010.974,352.925,-157.897,170.681,52.717,160.429
C02435=1010.981,353.172,-157.934,170.689,52.713,160.430
C02436=1010.987,353.420,-157.970,170.698,52.709,160.430
C02437=1010.996,353.718,-158.014,170.708,52.704,160.431
C02438=1011.005,354.015,-158.058,170.719,52.698,160.432
C02439=1011.013,354.312,-158.102,170.729,52.694,160.433
C02440=1011.021,354.609,-158.146,170.740,52.689,160.434
C02441=1011.028,354.857,-158.183,170.749,52.684,160.434
C02442=1011.036,355.104,-158.220,170.758,52.680,160.435
C02443=1011.042,355.351,-158.256,170.766,52.676,160.436
C02444=1011.049,355.598,-158.293,170.775,52.672,160.436
C02445=1011.057,355.846,-158.331,170.783,52.667,160.437
C02446=1011.064,356.092,-158.366,170.793,52.663,160.438
C02447=1011.071,356.340,-158.403,170.801,52.659,160.439
C02448=1011.078,356.587,-158.441,170.810,52.654,160.439
C02449=1011.085,356.834,-158.477,170.819,52.650,160.440
C02450=1011.092,357.081,-158.514,170.829,52.646,160.441
C02451=1011.099,357.328,-158.552,170.837,52.642,160.442
C02452=1011.106,357.576,-158.589,170.846,52.638,160.442
C02453=1011.114,357.822,-158.625,170.854,52.634,160.443
C02454=1011.121,358.070,-158.662,170.864,52.629,160.444
C02455=1011.128,358.317,-158.699,170.873,52.626,160.445
C02456=1011.135,358.564,-158.737,170.881,52.622,160.445
C02457=1011.142,358.811,-158.774,170.890,52.617,160.446
C02458=1011.149,359.058,-158.812,170.899,52.614,160.447
C02459=1011.156,359.305,-158.849,170.908,52.609,160.448
C02460=1011.164,359.552,-158.887,170.917,52.606,160.449
C02461=1011.171,359.799,-158.924,170.926,52.602,160.449
C02462=1011.178,360.047,-158.961,170.935,52.597,160.450
C02463=1011.185,360.293,-158.999,170.944,52.594,160.451
C02464=1011.193,360.541,-159.037,170.953,52.589,160.452
C02465=1011.200,360.788,-159.074,170.962,52.586,160.453
C02466=1011.207,361.035,-159.112,170.971,52.581,160.454
C02467=1011.214,361.282,-159.149,170.980,52.578,160.454
C02468=1011.222,361.529,-159.187,170.989,52.574,160.455
C02469=1011.229,361.776,-159.224,170.999,52.570,160.456
C02470=1011.236,362.023,-159.262,171.008,52.566,160.457
C02471=1011.243,362.271,-159.300,171.016,52.562,160.458
C02472=1011.251,362.517,-159.338,171.026,52.558,160.459
C02473=1011.258,362.764,-159.375,171.035,52.555,160.460
C02474=1011.265,363.011,-159.413,171.044,52.551,160.461
C02475=1011.273,363.258,-159.451,171.054,52.547,160.461
C02476=1011.280,363.505,-159.489,171.063,52.543,160.462
C02477=1011.288,363.753,-159.526,171.072,52.540,160.463
C02478=1011.296,363.999,-159.565,171.082,52.536,160.464
C02479=1011.303,364.246,-159.602,171.090,52.531,160.465
C02480=1011.310,364.493,-159.640,171.100,52.528,160.466
C02481=1011.318,364.762,-159.682,171.110,52.524,160.467
C02482=1011.326,365.030,-159.723,171.120,52.520,160.468
C02483=1011.335,365.298,-159.764,171.130,52.516,160.469
C02484=1011.343,365.566,-159.806,171.141,52.511,160.470
C02485=1011.350,365.813,-159.843,171.150,52.508,160.471
C02486=1011.358,366.060,-159.882,171.159,52.504,160.472
C02487=1011.366,366.308,-159.919,171.169,52.501,160.473
C02488=1011.373,366.554,-159.958,171.178,52.497,160.474
C02489=1011.381,366.801,-159.996,171.188,52.493,160.475
C02490=1011.388,367.048,-160.035,171.197,52.490,160.475
C02491=1011.396,367.295,-160.073,171.207,52.486,160.476
C02492=1011.403,367.541,-160.112,171.216,52.482,160.477
C02493=1011.411,367.789,-160.151,171.227,52.479,160.479
C02494=1011.418,368.035,-160.189,171.236,52.475,160.480
C02495=1011.426,368.282,-160.228,171.244,52.472,160.480
C02496=1011.433,368.529,-160.267,171.254,52.468,160.481
C02497=1011.445,368.888,-160.322,171.269,52.463,160.483
C02498=1011.455,369.247,-160.379,171.283,52.458,160.484
C02499=1011.466,369.606,-160.435,171.296,52.453,160.486
C02500=1011.478,369.965,-160.492,171.310,52.448,160.487
C02501=1011.485,370.212,-160.531,171.321,52.444,160.489
C02502=1011.493,370.458,-160.570,171.330,52.441,160.489
C02503=1011.501,370.705,-160.608,171.340,52.438,160.491
C02504=1011.508,370.952,-160.647,171.349,52.434,160.492
C02505=1011.517,371.199,-160.686,171.359,52.431,160.493
C02506=1011.525,371.446,-160.725,171.369,52.427,160.494
C02507=1011.532,371.693,-160.764,171.379,52.424,160.495
C02508=1011.540,371.939,-160.803,171.389,52.420,160.496
C02509=1011.548,372.187,-160.842,171.398,52.417,160.497
C02510=1011.555,372.433,-160.881,171.409,52.414,160.498
C02511=1011.563,372.680,-160.920,171.419,52.410,160.499
C02512=1011.572,372.927,-160.959,171.428,52.407,160.500
C02513=1011.580,373.173,-160.999,171.438,52.404,160.502
C02514=1011.587,373.420,-161.038,171.448,52.400,160.503
C02515=1011.596,373.667,-161.077,171.458,52.397,160.504
C02516=1011.603,373.913,-161.117,171.468,52.394,160.505
C02517=1011.267,371.818,-161.136,171.364,52.480,160.506
C02518=1011.260,371.570,-161.096,171.355,52.483,160.506
C02519=1011.252,371.323,-161.058,171.345,52.487,160.504
C02520=1011.244,371.077,-161.019,171.336,52.490,160.503
C02521=1011.236,370.830,-160.980,171.326,52.493,160.502
C02522=1011.229,370.583,-160.941,171.315,52.497,160.501
C02523=1011.220,370.337,-160.902,171.306,52.500,160.500
C02524=1011.214,370.090,-160.863,171.296,52.504,160.499
C02525=1011.205,369.843,-160.825,171.287,52.507,160.498
C02526=1011.196,369.532,-160.776,171.275,52.512,160.497
C02527=1011.186,369.220,-160.727,171.262,52.516,160.495
C02528=1011.177,368.909,-160.678,171.251,52.521,160.494
C02529=1011.168,368.598,-160.630,171.238,52.525,160.493
C02530=1011.159,368.351,-160.590,171.228,52.529,160.492
C02531=1011.152,368.105,-160.552,171.219,52.532,160.491
C02532=1011.144,367.857,-160.513,171.209,52.536,160.490
C02533=1011.137,367.610,-160.475,171.200,52.539,160.489
C02534=1011.129,367.364,-160.437,171.190,52.543,160.488
C02535=1011.122,367.116,-160.398,171.181,52.546,160.487
C02536=1011.115,366.870,-160.360,171.171,52.550,160.486
C02537=1011.107,366.623,-160.322,171.162,52.554,160.485
C02538=1011.100,366.376,-160.283,171.152,52.558,160.484
C02539=1011.092,366.128,-160.245,171.143,52.561,160.483
C02540=1011.085,365.882,-160.207,171.133,52.565,160.482
C02541=1011.077,365.635,-160.168,171.124,52.569,160.481
C02542=1011.069,365.387,-160.130,171.114,52.573,160.480
C02543=1011.062,365.141,-160.092,171.105,52.576,160.479
C02544=1011.055,364.894,-160.055,171.096,52.580,160.478
C02545=1011.047,364.647,-160.016,171.086,52.584,160.477
C02546=1011.040,364.400,-159.979,171.077,52.587,160.476
C02547=1011.032,364.152,-159.941,171.067,52.591,160.475
C02548=1011.024,363.906,-159.903,171.059,52.595,160.475
C02549=1011.017,363.659,-159.865,171.050,52.599,160.474
C02550=1011.010,363.412,-159.828,171.040,52.603,160.473
C02551=1011.002,363.165,-159.789,171.031,52.606,160.472
C02552=1010.995,362.918,-159.752,171.021,52.611,160.471
C02553=1010.988,362.671,-159.714,171.012,52.614,160.470
C02554=1010.981,362.424,-159.677,171.003,52.618,160.469
C02555=1010.973,362.177,-159.639,170.994,52.622,160.468
C02556=1010.966,361.930,-159.601,170.985,52.626,160.467
C02557=1010.959,361.683,-159.564,170.976,52.629,160.466
C02558=1010.951,361.436,-159.526,170.966,52.634,160.466
C02559=1010.944,361.189,-159.488,170.957,52.638,160.465
C02560=1010.937,360.941,-159.451,170.949,52.642,160.464
C02561=1010.930,360.694,-159.413,170.939,52.646,160.463
C02562=1010.922,360.447,-159.376,170.930,52.650,160.462
C02563=1010.915,360.200,-159.338,170.921,52.653,160.461
C02564=1010.908,359.953,-159.301,170.911,52.658,160.461
C02565=1010.901,359.706,-159.263,170.902,52.661,160.460
C02566=1010.893,359.459,-159.226,170.894,52.666,160.459
C02567=1010.886,359.212,-159.188,170.884,52.670,160.458
C02568=1010.879,358.965,-159.151,170.875,52.674,160.457
C02569=1010.872,358.718,-159.114,170.867,52.678,160.457
C02570=1010.865,358.470,-159.077,170.858,52.681,160.456
C02571=1010.858,358.223,-159.039,170.848,52.686,160.455
C02572=1010.851,357.976,-159.002,170.840,52.690,160.454
C02573=1010.844,357.729,-158.966,170.831,52.694,160.453
C02574=1010.837,357.482,-158.928,170.822,52.698,160.453
C02575=1010.829,357.235,-158.891,170.813,52.702,160.452
C02576=1010.822,356.987,-158.854,170.804,52.707,160.451
C02577=1010.815,356.741,-158.817,170.796,52.711,160.451
C02578=1010.808,356.493,-158.781,170.787,52.714,160.450
C02579=1010.801,356.246,-158.744,170.777,52.719,160.449
C02580=1010.794,355.999,-158.707,170.769,52.723,160.448
C02581=1010.787,355.752,-158.670,170.760,52.727,160.447
C02582=1010.780,355.505,-158.633,170.751,52.731,160.447
C02583=1010.773,355.257,-158.596,170.742,52.736,160.446
C02584=1010.765,355.010,-158.560,170.733,52.740,160.445
C02585=1010.759,354.763,-158.524,170.725,52.744,160.445
C02586=1010.750,354.442,-158.476,170.713,52.750,160.444
C02587=1010.741,354.121,-158.428,170.702,52.756,160.443
C02588=1010.732,353.800,-158.380,170.691,52.761,160.442
C02589=1010.723,353.479,-158.333,170.680,52.767,160.441
C02590=1010.715,353.232,-158.297,170.671,52.771,160.440
C02591=1010.709,352.985,-158.261,170.662,52.775,160.440
C02592=1010.702,352.737,-158.224,170.654,52.780,160.439
C02593=1010.695,352.490,-158.188,170.645,52.784,160.438
C02594=1010.688,352.243,-158.151,170.637,52.789,160.438
C02595=1010.681,351.996,-158.115,170.628,52.793,160.437
C02596=1010.674,351.748,-158.078,170.619,52.797,160.436
C02597=1010.667,351.501,-158.043,170.611,52.802,160.436
C02598=1010.661,351.254,-158.006,170.603,52.806,160.435
C02599=1010.653,351.006,-157.971,170.594,52.811,160.434
C02600=1010.647,350.759,-157.934,170.585,52.815,160.434
C02601=1010.640,350.513,-157.898,170.577,52.820,160.433
C02602=1010.633,350.265,-157.862,170.568,52.824,160.432
C02603=1010.626,350.017,-157.826,170.560,52.829,160.432
C02604=1010.620,349.770,-157.790,170.551,52.833,160.431
C02605=1010.612,349.523,-157.754,170.543,52.837,160.430
C02606=1010.606,349.275,-157.718,170.534,52.842,160.430
C02607=1010.599,349.028,-157.682,170.526,52.846,160.429
C02608=1010.593,348.781,-157.646,170.518,52.851,160.429
C02609=1010.585,348.533,-157.610,170.509,52.855,160.428
C02610=1010.579,348.286,-157.574,170.501,52.860,160.428
C02611=1010.572,348.039,-157.539,170.493,52.864,160.427
C02612=1010.566,347.792,-157.502,170.484,52.870,160.426
C02613=1010.559,347.544,-157.467,170.475,52.875,160.426
C02614=1010.553,347.296,-157.431,170.467,52.879,160.425
C02615=1010.546,347.049,-157.395,170.459,52.884,160.425
C02616=1010.540,346.802,-157.359,170.451,52.888,160.424
C02617=1010.532,346.555,-157.324,170.442,52.893,160.424
C02618=1010.526,346.308,-157.288,170.434,52.897,160.423
C02619=1010.520,346.060,-157.253,170.426,52.902,160.423
C02620=1010.513,345.813,-157.218,170.417,52.906,160.422
C02621=1010.507,345.566,-157.181,170.409,52.911,160.421
C02622=1010.500,345.318,-157.146,170.401,52.916,160.421
C02623=1010.493,345.071,-157.111,170.393,52.921,160.420
C02624=1010.486,344.823,-157.075,170.385,52.926,160.420
C02625=1010.480,344.575,-157.040,170.376,52.930,160.419
C02626=1010.473,344.328,-157.004,170.368,52.935,160.419
C02627=1010.466,344.080,-156.969,170.360,52.940,160.418
C02628=1010.459,343.833,-156.934,170.352,52.945,160.418
C02629=1010.454,343.586,-156.899,170.344,52.949,160.417
C02630=1010.447,343.339,-156.864,170.336,52.954,160.417
C02631=1010.440,343.091,-156.829,170.328,52.959,160.416
C02632=1010.434,342.844,-156.793,170.320,52.964,160.416
C02633=1010.427,342.596,-156.759,170.312,52.969,160.415
C02634=1010.421,342.348,-156.723,170.304,52.974,160.415
C02635=1010.414,342.101,-156.688,170.295,52.979,160.414
C02636=1010.408,341.853,-156.653,170.287,52.983,160.414
C02637=1010.401,341.606,-156.618,170.279,52.988,160.413
C02638=1010.396,341.359,-156.583,170.271,52.993,160.413
C02639=1010.389,341.111,-156.548,170.263,52.998,160.412
C02640=1010.382,340.864,-156.513,170.255,53.003,160.412
C02641=1010.375,340.616,-156.478,170.247,53.008,160.412
C02642=1010.369,340.368,-156.443,170.239,53.013,160.411
C02643=1010.363,340.122,-156.409,170.231,53.018,160.411
C02644=1010.357,339.873,-156.374,170.223,53.023,160.410
C02645=1010.350,339.626,-156.338,170.215,53.028,160.410
C02646=1010.342,339.303,-156.293,170.204,53.034,160.409
C02647=1010.333,338.979,-156.248,170.194,53.041,160.409
C02648=1010.326,338.656,-156.203,170.184,53.047,160.408
C02649=1010.317,338.332,-156.157,170.173,53.054,160.408
C02650=1010.311,338.085,-156.122,170.166,53.060,160.407
C02651=1010.305,337.838,-156.088,170.157,53.064,160.407
C02652=1010.298,337.590,-156.054,170.149,53.069,160.406
C02653=1010.291,337.342,-156.018,170.142,53.075,160.406
C02654=1010.286,337.095,-155.984,170.134,53.080,160.405
C02655=1010.279,336.847,-155.950,170.126,53.085,160.405
C02656=1010.272,336.599,-155.916,170.118,53.090,160.405
C02657=1010.266,336.352,-155.882,170.110,53.096,160.404
C02658=1010.260,336.104,-155.848,170.103,53.100,160.404
C02659=1010.254,335.857,-155.814,170.095,53.106,160.404
C02660=1010.247,335.610,-155.779,170.087,53.110,160.403
C02661=1010.241,335.362,-155.744,170.080,53.116,160.403
C02662=1010.235,335.114,-155.710,170.072,53.121,160.403
C02663=1010.229,334.867,-155.676,170.064,53.126,160.402
C02664=1010.222,334.619,-155.642,170.056,53.131,160.402
C02665=1010.216,334.372,-155.608,170.048,53.137,160.402
C02666=1010.209,334.124,-155.574,170.041,53.142,160.401
C02667=1010.203,333.877,-155.540,170.032,53.147,160.401
C02668=1010.197,333.628,-155.506,170.025,53.153,160.400
C02669=1010.191,333.381,-155.472,170.018,53.157,160.400
C02670=1010.186,333.134,-155.438,170.010,53.163,160.400
C02671=1010.179,332.886,-155.403,170.002,53.168,160.400
C02672=1010.173,332.638,-155.369,169.995,53.174,160.399
C02673=1010.167,332.391,-155.335,169.987,53.179,160.399
C02674=1010.161,332.143,-155.301,169.979,53.184,160.399
C02675=1010.155,331.895,-155.268,169.971,53.190,160.398
C02676=1010.149,331.648,-155.234,169.964,53.195,160.398
C02677=1010.142,331.400,-155.200,169.957,53.200,160.398
C02678=1010.137,331.152,-155.166,169.949,53.205,160.397
C02679=1010.130,330.905,-155.133,169.941,53.211,160.397
C02680=1010.124,330.657,-155.099,169.934,53.216,160.397
C02681=1010.118,330.409,-155.065,169.926,53.222,160.396
C02682=1010.112,330.162,-155.032,169.918,53.227,160.396
C02683=1010.106,329.915,-154.998,169.911,53.233,160.396
C02684=1010.100,329.666,-154.965,169.903,53.238,160.396
C02685=1010.093,329.419,-154.931,169.896,53.244,160.395
C02686=1010.088,329.171,-154.898,169.889,53.249,160.395
C02687=1010.082,328.924,-154.864,169.881,53.255,160.395
C02688=1010.075,328.676,-154.831,169.874,53.260,160.395
C02689=1010.069,328.428,-154.797,169.866,53.266,160.394
C02690=1010.063,328.181,-154.764,169.858,53.271,160.394
C02691=1010.057,327.933,-154.731,169.851,53.277,160.394
C02692=1010.052,327.685,-154.697,169.844,53.282,160.394
C02693=1010.045,327.438,-154.664,169.836,53.288,160.393
C02694=1010.039,327.190,-154.630,169.829,53.293,160.393
C02695=1010.034,326.942,-154.597,169.821,53.299,160.393
C02696=1010.028,326.694,-154.564,169.813,53.304,160.392
C02697=1010.022,326.447,-154.531,169.806,53.310,160.392
C02698=1010.016,326.199,-154.497,169.800,53.316,160.392
C02699=1010.010,325.952,-154.464,169.792,53.321,160.392
C02700=1010.004,325.704,-154.431,169.784,53.327,160.392
C02701=1009.998,325.456,-154.398,169.777,53.332,160.391
C02702=1009.993,325.208,-154.365,169.769,53.338,160.391
C02703=1009.986,324.961,-154.332,169.762,53.344,160.391
C02704=1009.980,324.713,-154.299,169.755,53.349,160.391
C02705=1009.974,324.465,-154.266,169.747,53.355,160.391
C02706=1009.966,324.138,-154.223,169.738,53.363,160.390
C02707=1009.958,323.809,-154.180,169.728,53.370,160.390
C02708=1009.950,323.482,-154.137,169.719,53.378,160.390
C02709=1009.942,323.154,-154.093,169.709,53.385,160.390
C02710=1009.936,322.906,-154.061,169.701,53.391,160.390
C02711=1009.930,322.658,-154.028,169.694,53.397,160.389
C02712=1009.923,322.411,-153.995,169.686,53.403,160.389
C02713=1009.917,322.162,-153.963,169.679,53.409,160.389
C02714=1009.912,321.914,-153.930,169.672,53.414,160.389
C02715=1009.907,321.667,-153.898,169.665,53.420,160.389
C02716=1009.900,321.419,-153.866,169.657,53.426,160.388
C02717=1009.894,321.172,-153.833,169.650,53.432,160.388
C02718=1009.888,320.924,-153.801,169.643,53.438,160.388
C02719=1009.882,320.676,-153.768,169.636,53.443,160.388
C02720=1009.876,320.427,-153.736,169.629,53.450,160.388
C02721=1009.871,320.181,-153.703,169.622,53.455,160.388
C02722=1009.865,319.932,-153.671,169.614,53.461,160.388
C02723=1009.859,319.684,-153.639,169.607,53.467,160.387
C02724=1009.852,319.437,-153.606,169.601,53.473,160.388
C02725=1009.848,319.189,-153.574,169.594,53.479,160.387
C02726=1009.842,318.941,-153.541,169.586,53.485,160.387
C02727=1009.836,318.693,-153.509,169.579,53.491,160.387
C02728=1009.830,318.445,-153.478,169.571,53.497,160.387
C02729=1009.824,318.198,-153.445,169.565,53.502,160.387
C02730=1009.818,317.950,-153.413,169.558,53.509,160.387
C02731=1009.813,317.702,-153.381,169.551,53.515,160.387
C02732=1009.807,317.454,-153.348,169.543,53.520,160.386
C02733=1009.802,317.207,-153.316,169.536,53.527,160.386
C02734=1009.796,316.958,-153.284,169.530,53.533,160.386
C02735=1009.790,316.710,-153.252,169.522,53.539,160.386
C02736=1009.784,316.463,-153.221,169.515,53.544,160.386
C02737=1009.779,316.215,-153.187,169.508,53.551,160.386
C02738=1009.773,315.967,-153.156,169.501,53.556,160.386
C02739=1009.767,315.719,-153.123,169.494,53.563,160.386
C02740=1009.762,315.472,-153.092,169.487,53.569,160.386
C02741=1009.756,315.223,-153.060,169.480,53.575,160.386
C02742=1009.751,314.976,-153.028,169.474,53.581,160.386
C02743=1009.745,314.727,-152.996,169.466,53.587,160.386
C02744=1009.740,314.480,-152.964,169.459,53.593,160.385
C02745=1009.734,314.232,-152.932,169.452,53.599,160.385
C02746=1009.729,313.984,-152.900,169.445,53.605,160.385
C02747=1009.723,313.737,-152.868,169.438,53.611,160.385
C02748=1009.717,313.488,-152.836,169.431,53.618,160.385
C02749=1009.712,313.241,-152.804,169.424,53.624,160.385
C02750=1009.707,312.992,-152.772,169.418,53.630,160.385
C02751=1009.701,312.745,-152.741,169.411,53.636,160.385
C02752=1009.696,312.497,-152.709,169.403,53.642,160.385
C02753=1009.690,312.249,-152.677,169.396,53.649,160.385
C02754=1009.684,312.002,-152.645,169.390,53.654,160.385
C02755=1009.680,311.754,-152.613,169.383,53.661,160.385
C02756=1009.674,311.506,-152.581,169.376,53.667,160.385
C02757=1009.668,311.258,-152.549,169.370,53.673,160.385
C02758=1009.663,311.010,-152.518,169.362,53.679,160.385
C02759=1009.658,310.762,-152.487,169.355,53.685,160.385
C02760=1009.652,310.514,-152.455,169.348,53.692,160.385
C02761=1009.647,310.266,-152.422,169.342,53.698,160.385
C02762=1009.642,310.018,-152.391,169.335,53.704,160.385
C02763=1009.637,309.771,-152.360,169.328,53.711,160.385
C02764=1009.631,309.523,-152.328,169.322,53.717,160.385
C02765=1009.626,309.274,-152.297,169.315,53.723,160.385
C02766=1009.619,308.953,-152.255,169.306,53.731,160.385
C02767=1009.612,308.630,-152.214,169.297,53.739,160.385
C02768=1009.605,308.308,-152.174,169.289,53.748,160.385
C02769=1009.598,307.987,-152.134,169.280,53.756,160.385
C02770=1009.592,307.738,-152.103,169.273,53.763,160.385
C02771=1009.586,307.490,-152.072,169.266,53.769,160.385
C02772=1009.581,307.242,-152.041,169.259,53.775,160.385
C02773=1009.575,306.995,-152.010,169.253,53.782,160.385
C02774=1009.570,306.746,-151.979,169.246,53.788,160.385
C02775=1009.564,306.499,-151.949,169.239,53.794,160.385
C02776=1009.559,306.250,-151.918,169.232,53.801,160.385
C02777=1009.553,306.002,-151.887,169.225,53.808,160.385
C02778=1009.547,305.754,-151.856,169.219,53.814,160.385
C02779=1009.542,305.507,-151.825,169.212,53.820,160.385
C02780=1009.537,305.258,-151.794,169.205,53.827,160.385
C02781=1009.531,305.011,-151.764,169.198,53.834,160.385
C02782=1009.526,304.763,-151.733,169.193,53.840,160.386
C02783=1009.520,304.515,-151.703,169.185,53.847,160.385
C02784=1009.515,304.267,-151.672,169.179,53.853,160.386
C02785=1009.509,304.019,-151.641,169.172,53.860,160.386
C02786=1009.504,303.771,-151.610,169.166,53.866,160.386
C02787=1009.498,303.523,-151.580,169.159,53.873,160.386
C02788=1009.493,303.274,-151.550,169.152,53.880,160.386
C02789=1009.487,303.026,-151.519,169.146,53.886,160.386
C02790=1009.482,302.778,-151.488,169.139,53.893,160.386
C02791=1009.477,302.530,-151.458,169.132,53.900,160.386
C02792=1009.471,302.282,-151.427,169.125,53.906,160.386
C02793=1009.466,302.034,-151.397,169.120,53.912,160.386
C02794=1009.461,301.786,-151.366,169.113,53.919,160.387
C02795=1009.455,301.538,-151.336,169.106,53.926,160.386
C02796=1009.450,301.290,-151.305,169.099,53.933,160.387
C02797=1009.445,301.042,-151.275,169.093,53.939,160.387
C02798=1009.440,300.794,-151.244,169.086,53.946,160.387
C02799=1009.434,300.546,-151.215,169.080,53.953,160.387
C02800=1009.429,300.298,-151.184,169.074,53.959,160.387
C02801=1009.424,300.050,-151.153,169.067,53.965,160.387
C02802=1009.418,299.802,-151.123,169.060,53.972,160.387
C02803=1009.414,299.554,-151.093,169.053,53.979,160.387
C02804=1009.408,299.306,-151.062,169.048,53.986,160.388
C02805=1009.403,299.057,-151.032,169.041,53.992,160.387
C02806=1009.398,298.809,-151.002,169.034,53.999,160.388
C02807=1009.393,298.561,-150.971,169.028,54.006,160.388
C02808=1009.388,298.314,-150.942,169.022,54.013,160.388
C02809=1009.383,298.065,-150.911,169.015,54.020,160.388
C02810=1009.377,297.817,-150.881,169.009,54.026,160.388
C02811=1009.372,297.569,-150.850,169.002,54.033,160.388
C02812=1009.367,297.321,-150.821,168.995,54.040,160.388
C02813=1009.362,297.073,-150.790,168.989,54.047,160.389
C02814=1009.354,296.694,-150.744,168.979,54.057,160.389
C02815=1009.346,296.315,-150.698,168.970,54.068,160.389
C02816=1009.339,295.935,-150.652,168.960,54.078,160.389
C02817=1009.331,295.557,-150.606,168.950,54.089,160.389
C02818=1009.091,296.452,-151.080,168.948,54.121,160.397
C02819=1009.099,296.863,-151.130,168.959,54.110,160.396
C02820=1009.107,297.274,-151.179,168.970,54.098,160.396
C02821=1009.116,297.685,-151.230,168.981,54.088,160.396
C02822=1009.124,298.096,-151.279,168.991,54.077,160.396
C02823=1009.129,298.344,-151.310,168.998,54.070,160.396
C02824=1009.135,298.592,-151.340,169.004,54.063,160.396
C02825=1009.139,298.840,-151.370,169.010,54.056,160.395
C02826=1009.145,299.088,-151.400,169.017,54.050,160.395
C02827=1009.150,299.336,-151.431,169.024,54.043,160.395
C02828=1009.156,299.584,-151.461,169.030,54.036,160.395
C02829=1009.160,299.832,-151.491,169.036,54.029,160.395
C02830=1009.166,300.080,-151.521,169.043,54.023,160.395
C02831=1009.170,300.329,-151.552,169.050,54.016,160.395
C02832=1009.176,300.577,-151.582,169.056,54.009,160.395
C02833=1009.181,300.825,-151.613,169.063,54.003,160.395
C02834=1009.187,301.073,-151.643,169.069,53.996,160.395
C02835=1009.191,301.321,-151.673,169.077,53.990,160.395
C02836=1009.197,301.569,-151.704,169.082,53.983,160.394
C02837=1009.202,301.817,-151.735,169.089,53.976,160.394
C02838=1009.208,302.065,-151.764,169.096,53.970,160.394
C02839=1009.213,302.313,-151.795,169.102,53.963,160.394
C02840=1009.218,302.561,-151.825,169.109,53.957,160.394
C02841=1009.224,302.809,-151.856,169.116,53.950,160.394
C02842=1009.229,303.057,-151.887,169.122,53.943,160.394
C02843=1009.234,303.306,-151.917,169.128,53.937,160.394
C02844=1009.239,303.553,-151.947,169.135,53.930,160.394
C02845=1009.244,303.801,-151.978,169.142,53.924,160.394
C02846=1009.250,304.049,-152.008,169.149,53.917,160.394
C02847=1009.255,304.297,-152.039,169.155,53.911,160.394
C02848=1009.261,304.545,-152.070,169.162,53.904,160.394
C02849=1009.266,304.793,-152.100,169.169,53.897,160.394
C02850=1009.272,305.041,-152.131,169.176,53.890,160.394
C02851=1009.277,305.289,-152.162,169.182,53.884,160.393
C02852=1009.284,305.537,-152.193,169.189,53.878,160.394
C02853=1009.289,305.786,-152.223,169.196,53.871,160.393
C02854=1009.294,306.033,-152.254,169.203,53.865,160.394
C02855=1009.300,306.282,-152.285,169.208,53.858,160.393
C02856=1009.305,306.530,-152.316,169.216,53.852,160.393
C02857=1009.310,306.777,-152.346,169.223,53.846,160.393
C02858=1009.316,307.026,-152.377,169.229,53.839,160.393
C02859=1009.321,307.273,-152.407,169.236,53.833,160.393
C02860=1009.327,307.521,-152.439,169.243,53.827,160.393
C02861=1009.333,307.769,-152.469,169.249,53.820,160.393
C02862=1009.338,308.018,-152.501,169.257,53.813,160.393
C02863=1009.346,308.342,-152.541,169.265,53.805,160.393
C02864=1009.353,308.666,-152.582,169.275,53.797,160.393
C02865=1009.360,308.990,-152.623,169.283,53.788,160.393
C02866=1009.366,309.314,-152.664,169.292,53.781,160.393
C02867=1009.372,309.563,-152.695,169.299,53.774,160.393
C02868=1009.377,309.810,-152.727,169.306,53.768,160.393
C02869=1009.382,310.059,-152.759,169.313,53.762,160.393
C02870=1009.387,310.307,-152.791,169.319,53.755,160.393
C02871=1009.393,310.554,-152.822,169.326,53.749,160.393
C02872=1009.398,310.802,-152.854,169.333,53.743,160.393
C02873=1009.403,311.050,-152.885,169.339,53.737,160.393
C02874=1009.409,311.298,-152.917,169.346,53.730,160.393
C02875=1009.414,311.546,-152.949,169.354,53.724,160.394
C02876=1009.419,311.793,-152.981,169.361,53.718,160.394
C02877=1009.424,312.042,-153.012,169.367,53.712,160.394
C02878=1009.430,312.290,-153.044,169.374,53.706,160.394
C02879=1009.436,312.537,-153.075,169.381,53.699,160.394
C02880=1009.441,312.785,-153.107,169.387,53.693,160.394
C02881=1009.446,313.033,-153.140,169.395,53.687,160.394
C02882=1009.452,313.281,-153.171,169.402,53.681,160.394
C02883=1009.457,313.528,-153.203,169.409,53.675,160.394
C02884=1009.463,313.777,-153.235,169.415,53.669,160.394
C02885=1009.468,314.024,-153.267,169.423,53.663,160.394
C02886=1009.474,314.272,-153.299,169.430,53.657,160.394
C02887=1009.479,314.520,-153.331,169.437,53.651,160.394
C02888=1009.484,314.768,-153.363,169.443,53.645,160.394
C02889=1009.490,315.016,-153.395,169.450,53.639,160.394
C02890=1009.496,315.263,-153.426,169.458,53.632,160.394
C02891=1009.502,315.512,-153.458,169.465,53.626,160.394
C02892=1009.507,315.759,-153.490,169.471,53.621,160.395
C02893=1009.512,316.008,-153.523,169.479,53.615,160.395
C02894=1009.518,316.255,-153.554,169.486,53.608,160.395
C02895=1009.524,316.503,-153.586,169.493,53.602,160.395
C02896=1009.529,316.751,-153.618,169.500,53.596,160.395
C02897=1009.535,316.999,-153.650,169.507,53.591,160.395
C02898=1009.541,317.246,-153.682,169.514,53.584,160.395
C02899=1009.546,317.495,-153.715,169.521,53.578,160.395
C02900=1009.552,317.743,-153.747,169.529,53.572,160.396
C02901=1009.557,317.990,-153.779,169.535,53.567,160.396
C02902=1009.564,318.238,-153.811,169.542,53.560,160.396
C02903=1009.569,318.485,-153.843,169.550,53.555,160.396
C02904=1009.575,318.734,-153.875,169.557,53.549,160.396
C02905=1009.581,318.981,-153.908,169.564,53.542,160.396
C02906=1009.586,319.229,-153.940,169.571,53.537,160.396
C02907=1009.592,319.477,-153.972,169.578,53.531,160.396
C02908=1009.598,319.725,-154.005,169.585,53.525,160.396
C02909=1009.604,319.972,-154.037,169.593,53.519,160.397
C02910=1009.610,320.221,-154.069,169.600,53.513,160.397
C02911=1009.615,320.468,-154.102,169.607,53.507,160.397
C02912=1009.621,320.717,-154.134,169.614,53.501,160.397
C02913=1009.627,320.964,-154.166,169.621,53.496,160.397
C02914=1009.633,321.212,-154.198,169.628,53.490,160.397
C02915=1009.639,321.459,-154.231,169.636,53.484,160.398
C02916=1009.644,321.708,-154.264,169.643,53.478,160.398
C02917=1009.651,321.955,-154.296,169.651,53.472,160.398
C02918=1009.656,322.203,-154.328,169.657,53.466,160.398
C02919=1009.662,322.451,-154.361,169.665,53.461,160.398
C02920=1009.669,322.698,-154.394,169.672,53.454,160.398
C02921=1009.675,322.946,-154.426,169.680,53.449,160.399
C02922=1009.680,323.194,-154.459,169.687,53.443,160.399
C02923=1009.688,323.525,-154.502,169.697,53.435,160.399
C02924=1009.696,323.854,-154.546,169.706,53.428,160.399
C02925=1009.704,324.185,-154.589,169.716,53.420,160.399
C02926=1009.713,324.515,-154.632,169.726,53.413,160.400
C02927=1009.719,324.763,-154.665,169.733,53.406,160.400
C02928=1009.725,325.011,-154.698,169.741,53.401,160.400
C02929=1009.731,325.258,-154.731,169.748,53.395,160.401
C02930=1009.736,325.506,-154.764,169.755,53.390,160.401
C02931=1009.743,325.754,-154.797,169.763,53.385,160.401
C02932=1009.748,326.002,-154.830,169.770,53.378,160.401
C02933=1009.754,326.249,-154.864,169.778,53.373,160.401
C02934=1009.760,326.496,-154.897,169.785,53.367,160.402
C02935=1009.766,326.744,-154.930,169.793,53.362,160.402
C02936=1009.772,326.992,-154.963,169.800,53.357,160.402
C02937=1009.778,327.240,-154.996,169.807,53.351,160.402
C02938=1009.783,327.488,-155.030,169.815,53.345,160.403
C02939=1009.790,327.735,-155.063,169.822,53.340,160.403
C02940=1009.795,327.983,-155.097,169.830,53.334,160.403
C02941=1009.801,328.231,-155.130,169.838,53.329,160.404
C02942=1009.807,328.478,-155.163,169.845,53.323,160.404
C02943=1009.813,328.725,-155.197,169.852,53.318,160.404
C02944=1009.819,328.973,-155.229,169.860,53.313,160.404
C02945=1009.826,329.222,-155.263,169.867,53.307,160.405
C02946=1009.831,329.469,-155.297,169.875,53.301,160.405
C02947=1009.838,329.716,-155.330,169.883,53.296,160.405
C02948=1009.844,329.964,-155.364,169.890,53.290,160.405
C02949=1009.849,330.212,-155.397,169.898,53.285,160.406
C02950=1009.856,330.460,-155.430,169.906,53.279,160.406
C02951=1009.862,330.707,-155.465,169.912,53.274,160.406
C02952=1009.868,330.955,-155.498,169.920,53.269,160.406
C02953=1009.874,331.202,-155.531,169.927,53.263,160.407
C02954=1009.880,331.449,-155.565,169.936,53.258,160.407
C02955=1009.886,331.698,-155.599,169.943,53.253,160.407
C02956=1009.892,331.945,-155.633,169.951,53.247,160.408
C02957=1009.899,332.192,-155.667,169.958,53.241,160.408
C02958=1009.905,332.441,-155.700,169.967,53.237,160.409
C02959=1009.911,332.688,-155.734,169.974,53.231,160.409
C02960=1009.916,332.935,-155.768,169.981,53.226,160.409
C02961=1009.923,333.183,-155.803,169.989,53.221,160.409
C02962=1009.929,333.431,-155.837,169.997,53.216,160.410
C02963=1009.935,333.678,-155.871,170.004,53.210,160.410
C02964=1009.941,333.927,-155.905,170.012,53.205,160.411
C02965=1009.947,334.174,-155.939,170.020,53.200,160.411
C02966=1009.953,334.422,-155.973,170.028,53.194,160.411
C02967=1009.960,334.669,-156.007,170.036,53.189,160.412
C02968=1009.966,334.917,-156.041,170.043,53.184,160.412
C02969=1009.972,335.164,-156.075,170.052,53.179,160.412
C02970=1009.978,335.411,-156.109,170.059,53.173,160.413
C02971=1009.984,335.659,-156.144,170.067,53.168,160.413
C02972=1009.990,335.907,-156.178,170.074,53.163,160.413
C02973=1009.997,336.155,-156.212,170.082,53.158,160.414
C02974=1010.003,336.403,-156.246,170.090,53.153,160.414
C02975=1010.009,336.650,-156.280,170.098,53.148,160.415
C02976=1010.017,336.897,-156.315,170.105,53.142,160.415
C02977=1010.022,337.144,-156.349,170.114,53.138,160.415
C02978=1010.029,337.392,-156.383,170.121,53.132,160.416
C02979=1010.035,337.640,-156.418,170.129,53.127,160.416
C02980=1010.041,337.888,-156.452,170.137,53.122,160.417
C02981=1010.048,338.135,-156.487,170.145,53.117,160.417
C02982=1010.054,338.382,-156.521,170.153,53.112,160.417
C02983=1010.062,338.708,-156.567,170.164,53.105,160.418
C02984=1010.070,339.033,-156.613,170.174,53.098,160.419
C02985=1010.078,339.360,-156.658,170.184,53.092,160.419
C02986=1010.087,339.686,-156.704,170.195,53.085,160.420
C02987=1010.093,339.933,-156.739,170.203,53.081,160.420
C02988=1010.100,340.181,-156.773,170.211,53.076,160.421
C02989=1010.106,340.428,-156.808,170.219,53.071,160.421
C02990=1010.112,340.675,-156.844,170.227,53.065,160.421
C02991=1010.118,340.923,-156.878,170.235,53.060,160.422
C02992=1010.125,341.170,-156.913,170.243,53.056,160.422
C02993=1010.132,341.418,-156.949,170.251,53.051,160.423
C02994=1010.138,341.666,-156.983,170.259,53.046,160.423
C02995=1010.144,341.912,-157.018,170.267,53.041,160.424
C02996=1010.150,342.160,-157.053,170.275,53.036,160.424
C02997=1010.157,342.407,-157.089,170.283,53.031,160.425
C02998=1010.164,342.655,-157.123,170.291,53.026,160.425
C02999=1010.170,342.903,-157.158,170.300,53.022,160.426
C03000=1010.177,343.150,-157.194,170.308,53.017,160.426
C03001=1010.183,343.398,-157.229,170.316,53.012,160.427
C03002=1010.190,343.645,-157.264,170.324,53.007,160.427
C03003=1010.197,343.892,-157.299,170.332,53.002,160.428
C03004=1010.202,344.139,-157.335,170.340,52.997,160.428
C03005=1010.209,344.387,-157.370,170.348,52.992,160.429
C03006=1010.216,344.634,-157.405,170.357,52.988,160.429
C03007=1010.223,344.882,-157.440,170.366,52.983,160.430
C03008=1010.229,345.129,-157.476,170.374,52.978,160.430
C03009=1010.235,345.377,-157.511,170.382,52.973,160.431
C03010=1010.243,345.625,-157.546,170.390,52.968,160.431
C03011=1010.249,345.872,-157.582,170.399,52.964,160.432
C03012=1010.256,346.120,-157.617,170.407,52.959,160.433
C03013=1010.262,346.367,-157.652,170.415,52.955,160.433
C03014=1010.269,346.614,-157.689,170.423,52.950,160.434
C03015=1010.275,346.861,-157.724,170.432,52.946,160.434
C03016=1010.281,347.109,-157.760,170.440,52.941,160.435
C03017=1010.288,347.356,-157.796,170.448,52.936,160.436
C03018=1010.295,347.603,-157.831,170.456,52.932,160.436
C03019=1010.302,347.850,-157.867,170.464,52.927,160.436
C03020=1010.309,348.098,-157.903,170.473,52.923,160.437
C03021=1010.315,348.346,-157.938,170.482,52.917,160.438
C03022=1010.322,348.593,-157.974,170.491,52.913,160.439
C03023=1010.328,348.840,-158.010,170.499,52.908,160.439
C03024=1010.335,349.087,-158.046,170.507,52.904,160.440
C03025=1010.342,349.335,-158.083,170.515,52.899,160.440
C03026=1010.349,349.582,-158.118,170.524,52.895,160.441
C03027=1010.355,349.829,-158.154,170.532,52.890,160.441
C03028=1010.362,350.077,-158.189,170.541,52.886,160.442
C03029=1010.369,350.325,-158.226,170.550,52.881,160.443
C03030=1010.376,350.571,-158.262,170.558,52.877,160.443
C03031=1010.382,350.819,-158.298,170.567,52.872,160.444
C03032=1010.390,351.066,-158.334,170.575,52.868,160.445
C03033=1010.396,351.313,-158.370,170.583,52.863,160.445
C03034=1010.403,351.560,-158.406,170.592,52.859,160.446
C03035=1010.410,351.808,-158.443,170.600,52.855,160.447
C03036=1010.417,352.055,-158.478,170.610,52.850,160.447
C03037=1010.424,352.303,-158.515,170.618,52.846,160.448
C03038=1010.431,352.550,-158.551,170.627,52.841,160.449
C03039=1010.437,352.797,-158.587,170.635,52.837,160.449
C03040=1010.444,353.045,-158.624,170.644,52.833,160.450
C03041=1010.451,353.291,-158.660,170.653,52.828,160.451
C03042=1010.458,353.539,-158.697,170.661,52.824,160.451
C03043=1010.467,353.863,-158.745,170.673,52.818,160.452
C03044=1010.476,354.185,-158.793,170.684,52.812,160.453
C03045=1010.486,354.508,-158.840,170.696,52.807,160.454
C03046=1010.495,354.832,-158.888,170.707,52.801,160.455
C03047=1010.501,355.079,-158.925,170.716,52.797,160.456
C03048=1010.508,355.326,-158.962,170.724,52.793,160.457
C03049=1010.515,355.573,-158.998,170.734,52.788,160.457
C03050=1010.522,355.820,-159.035,170.742,52.784,160.458
C03051=1010.529,356.068,-159.072,170.751,52.780,160.459
C03052=1010.536,356.314,-159.108,170.759,52.776,160.459
C03053=1010.543,356.562,-159.145,170.769,52.771,160.460
C03054=1010.551,356.809,-159.182,170.777,52.767,160.461
C03055=1010.557,357.056,-159.219,170.786,52.764,160.462
C03056=1010.565,357.303,-159.256,170.795,52.759,160.463
C03057=1010.572,357.551,-159.293,170.805,52.755,160.463
C03058=1010.579,357.798,-159.330,170.813,52.751,160.464
C03059=1010.585,358.045,-159.367,170.822,52.746,160.465
C03060=1010.593,358.292,-159.404,170.832,52.743,160.466
C03061=1010.601,358.539,-159.441,170.840,52.738,160.466
C03062=1010.608,358.787,-159.478,170.849,52.734,160.467
C03063=1010.614,359.033,-159.515,170.858,52.731,160.468
C03064=1010.622,359.280,-159.553,170.867,52.726,160.469
C03065=1010.629,359.527,-159.590,170.876,52.723,160.470
C03066=1010.635,359.775,-159.628,170.885,52.718,160.470
C03067=1010.643,360.022,-159.666,170.895,52.714,160.472
C03068=1010.650,360.269,-159.703,170.903,52.710,160.472
C03069=1010.656,360.516,-159.740,170.912,52.707,160.473
C03070=1010.663,360.763,-159.777,170.922,52.702,160.474
C03071=1010.671,361.010,-159.815,170.931,52.699,160.475
C03072=1010.678,361.257,-159.853,170.939,52.694,160.476
C03073=1010.685,361.504,-159.891,170.949,52.690,160.477
C03074=1010.693,361.751,-159.928,170.958,52.686,160.477
C03075=1010.700,361.998,-159.966,170.967,52.683,160.478
C03076=1010.707,362.246,-160.003,170.977,52.679,160.479
C03077=1010.714,362.493,-160.041,170.985,52.675,160.480
C03078=1010.722,362.740,-160.078,170.994,52.671,160.481
C03079=1010.729,362.987,-160.116,171.004,52.667,160.482
C03080=1010.736,363.233,-160.154,171.013,52.664,160.483
C03081=1010.744,363.481,-160.191,171.023,52.659,160.483
C03082=1010.751,363.728,-160.229,171.032,52.655,160.484
C03083=1010.759,363.975,-160.268,171.041,52.652,160.485
C03084=1010.766,364.222,-160.305,171.051,52.648,160.486
C03085=1010.774,364.469,-160.343,171.060,52.644,160.487
C03086=1010.781,364.716,-160.381,171.069,52.640,160.488
C03087=1010.788,364.963,-160.418,171.078,52.636,160.489
C03088=1010.796,365.209,-160.457,171.088,52.632,160.490
C03089=1010.804,365.457,-160.495,171.097,52.629,160.491
C03090=1010.811,365.704,-160.533,171.107,52.625,160.492
C03091=1010.819,365.951,-160.570,171.116,52.621,160.493
C03092=1010.826,366.197,-160.609,171.126,52.618,160.494
C03093=1010.834,366.445,-160.646,171.135,52.614,160.495
C03094=1010.841,366.692,-160.685,171.145,52.610,160.496
C03095=1010.849,366.938,-160.723,171.154,52.606,160.497
C03096=1010.856,367.186,-160.762,171.164,52.603,160.498
C03097=1010.864,367.432,-160.800,171.174,52.600,160.499
C03098=1010.871,367.679,-160.838,171.184,52.596,160.500
C03099=1010.878,367.926,-160.877,171.192,52.592,160.501
C03100=1010.886,368.173,-160.915,171.202,52.588,160.502
C03101=1010.894,368.420,-160.954,171.212,52.585,160.503
C03102=1010.901,368.667,-160.993,171.222,52.581,160.504
C03103=1010.909,368.932,-161.034,171.232,52.577,160.505
C03104=1010.918,369.197,-161.075,171.242,52.574,160.506
C03105=1010.926,369.462,-161.117,171.252,52.570,160.507
C03106=1010.934,369.727,-161.159,171.263,52.566,160.508
C03107=1010.602,367.628,-161.183,171.161,52.653,160.510
C03108=1010.595,367.381,-161.145,171.152,52.657,160.509
C03109=1010.587,367.135,-161.107,171.142,52.661,160.508
C03110=1010.581,366.888,-161.068,171.134,52.664,160.507
C03111=1010.572,366.641,-161.030,171.124,52.668,160.506
C03112=1010.565,366.394,-160.991,171.114,52.671,160.505
C03113=1010.558,366.147,-160.954,171.104,52.675,160.504
C03114=1010.550,365.901,-160.916,171.095,52.679,160.503
C03115=1010.542,365.653,-160.878,171.085,52.683,160.502
C03116=1010.535,365.406,-160.840,171.076,52.686,160.501
C03117=1010.527,365.159,-160.802,171.067,52.691,160.500
C03118=1010.520,364.912,-160.764,171.058,52.694,160.499
C03119=1010.513,364.665,-160.726,171.048,52.698,160.498
C03120=1010.505,364.418,-160.688,171.039,52.702,160.498
C03121=1010.497,364.171,-160.650,171.029,52.706,160.496
C03122=1010.490,363.924,-160.613,171.020,52.709,160.496
C03123=1010.483,363.677,-160.575,171.010,52.713,160.495
C03124=1010.476,363.430,-160.538,171.001,52.717,160.494
C03125=1010.468,363.183,-160.499,170.992,52.721,160.493
C03126=1010.461,362.936,-160.462,170.982,52.725,160.492
C03127=1010.453,362.689,-160.424,170.973,52.728,160.491
C03128=1010.446,362.442,-160.387,170.964,52.733,160.490
C03129=1010.439,362.195,-160.349,170.955,52.737,160.489
C03130=1010.432,361.947,-160.312,170.946,52.740,160.488
C03131=1010.424,361.700,-160.274,170.936,52.745,160.488
C03132=1010.417,361.453,-160.237,170.927,52.748,160.487
C03133=1010.410,361.206,-160.199,170.917,52.752,160.486
C03134=1010.403,360.959,-160.162,170.909,52.756,160.485
C03135=1010.396,360.712,-160.124,170.900,52.760,160.484
C03136=1010.388,360.465,-160.086,170.890,52.765,160.483
C03137=1010.382,360.218,-160.049,170.881,52.768,160.482
C03138=1010.374,359.971,-160.012,170.873,52.772,160.482
C03139=1010.367,359.724,-159.974,170.863,52.776,160.481
C03140=1010.360,359.477,-159.937,170.854,52.780,160.480
C03141=1010.353,359.230,-159.899,170.846,52.785,160.479
C03142=1010.346,358.983,-159.863,170.836,52.789,160.478
C03143=1010.339,358.735,-159.825,170.827,52.793,160.477
C03144=1010.332,358.488,-159.788,170.818,52.796,160.476
C03145=1010.325,358.241,-159.750,170.809,52.800,160.476
C03146=1010.318,357.994,-159.714,170.800,52.805,160.475
C03147=1010.311,357.747,-159.676,170.791,52.809,160.474
C03148=1010.304,357.499,-159.639,170.782,52.813,160.473
C03149=1010.297,357.252,-159.602,170.773,52.817,160.473
C03150=1010.290,357.005,-159.566,170.764,52.822,160.472
C03151=1010.283,356.758,-159.529,170.756,52.826,160.471
C03152=1010.276,356.510,-159.492,170.747,52.829,160.470
C03153=1010.268,356.264,-159.456,170.737,52.834,160.469
C03154=1010.261,356.017,-159.418,170.729,52.838,160.469
C03155=1010.255,355.770,-159.382,170.720,52.842,160.468
C03156=1010.248,355.522,-159.345,170.711,52.847,160.467
C03157=1010.240,355.274,-159.309,170.702,52.851,160.466
C03158=1010.234,355.028,-159.272,170.694,52.855,160.466
C03159=1010.227,354.780,-159.235,170.685,52.859,160.465
C03160=1010.219,354.485,-159.192,170.674,52.864,160.464
C03161=1010.211,354.189,-159.148,170.664,52.869,160.463
C03162=1010.201,353.894,-159.104,170.654,52.875,160.463
C03163=1010.193,353.598,-159.061,170.643,52.880,160.462
C03164=1010.187,353.351,-159.025,170.634,52.885,160.461
C03165=1010.180,353.103,-158.988,170.625,52.889,160.460
C03166=1010.173,352.857,-158.952,170.617,52.893,160.459
C03167=1010.166,352.609,-158.915,170.608,52.897,160.459
C03168=1010.160,352.362,-158.879,170.600,52.902,160.458
C03169=1010.153,352.115,-158.843,170.590,52.907,160.457
C03170=1010.146,351.867,-158.806,170.582,52.911,160.457
C03171=1010.139,351.620,-158.771,170.573,52.915,160.456
C03172=1010.133,351.373,-158.734,170.565,52.920,160.456
C03173=1010.125,351.125,-158.698,170.557,52.924,160.455
C03174=1010.119,350.878,-158.662,170.548,52.928,160.454
C03175=1010.112,350.631,-158.627,170.539,52.934,160.454
C03176=1010.105,350.383,-158.590,170.530,52.938,160.453
C03177=1010.098,350.136,-158.555,170.522,52.942,160.452
C03178=1010.092,349.889,-158.518,170.514,52.947,160.452
C03179=1010.085,349.642,-158.482,170.505,52.951,160.451
C03180=1010.078,349.394,-158.446,170.497,52.956,160.450
C03181=1010.071,349.147,-158.410,170.488,52.960,160.450
C03182=1010.064,348.900,-158.375,170.480,52.965,160.449
C03183=1010.058,348.653,-158.339,170.471,52.970,160.448
C03184=1010.051,348.405,-158.304,170.463,52.974,160.448
C03185=1010.044,348.157,-158.267,170.454,52.979,160.447
C03186=1010.037,347.910,-158.232,170.446,52.983,160.447
C03187=1010.031,347.662,-158.196,170.438,52.988,160.446
C03188=1010.024,347.416,-158.160,170.430,52.993,160.446
C03189=1010.018,347.168,-158.124,170.421,52.997,160.445
C03190=1010.012,346.921,-158.089,170.412,53.002,160.444
C03191=1010.005,346.674,-158.053,170.404,53.007,160.444
C03192=1009.998,346.426,-158.018,170.395,53.011,160.443
C03193=1009.992,346.179,-157.982,170.387,53.016,160.442
C03194=1009.986,345.931,-157.947,170.379,53.021,160.442
C03195=1009.980,345.684,-157.911,170.371,53.025,160.441
C03196=1009.973,345.437,-157.875,170.362,53.030,160.441
C03197=1009.966,345.189,-157.840,170.354,53.035,160.440
C03198=1009.959,344.942,-157.805,170.346,53.040,160.440
C03199=1009.952,344.695,-157.770,170.338,53.044,160.439
C03200=1009.946,344.447,-157.734,170.330,53.049,160.439
C03201=1009.940,344.199,-157.700,170.322,53.053,160.438
C03202=1009.933,343.952,-157.665,170.313,53.058,160.438
C03203=1009.926,343.704,-157.629,170.305,53.063,160.437
C03204=1009.920,343.457,-157.594,170.296,53.068,160.437
C03205=1009.913,343.209,-157.559,170.288,53.073,160.436
C03206=1009.907,342.962,-157.523,170.280,53.078,160.436
C03207=1009.900,342.715,-157.488,170.272,53.083,160.435
C03208=1009.895,342.467,-157.454,170.264,53.088,160.435
C03209=1009.888,342.220,-157.418,170.256,53.093,160.434
C03210=1009.881,341.972,-157.383,170.248,53.098,160.434
C03211=1009.874,341.725,-157.348,170.240,53.103,160.433
C03212=1009.868,341.477,-157.314,170.231,53.107,160.433
C03213=1009.863,341.230,-157.278,170.223,53.112,160.432
C03214=1009.856,340.982,-157.244,170.215,53.117,160.432
C03215=1009.849,340.735,-157.209,170.207,53.122,160.431
C03216=1009.843,340.487,-157.174,170.199,53.127,160.431
C03217=1009.837,340.240,-157.140,170.191,53.132,160.430
C03218=1009.830,339.993,-157.105,170.183,53.137,160.430
C03219=1009.824,339.744,-157.070,170.175,53.142,160.429
C03220=1009.815,339.417,-157.024,170.165,53.149,160.429
C03221=1009.808,339.089,-156.978,170.154,53.156,160.428
C03222=1009.799,338.760,-156.932,170.144,53.162,160.428
C03223=1009.791,338.432,-156.886,170.134,53.169,160.427
C03224=1009.784,338.185,-156.851,170.125,53.174,160.427
C03225=1009.779,337.937,-156.817,170.117,53.178,160.426
C03226=1009.772,337.689,-156.783,170.109,53.183,160.426
C03227=1009.766,337.442,-156.748,170.102,53.189,160.425
C03228=1009.759,337.195,-156.713,170.094,53.194,160.425
C03229=1009.754,336.947,-156.679,170.086,53.199,160.424
C03230=1009.747,336.699,-156.645,170.078,53.204,160.424
C03231=1009.741,336.453,-156.611,170.070,53.209,160.423
C03232=1009.734,336.205,-156.577,170.062,53.215,160.423
C03233=1009.728,335.957,-156.543,170.054,53.219,160.423
C03234=1009.722,335.709,-156.509,170.046,53.225,160.422
C03235=1009.716,335.462,-156.474,170.038,53.230,160.422
C03236=1009.709,335.214,-156.440,170.031,53.235,160.422
C03237=1009.704,334.967,-156.406,170.022,53.240,160.421
C03238=1009.697,334.719,-156.372,170.015,53.246,160.421
C03239=1009.691,334.471,-156.338,170.007,53.251,160.421
C03240=1009.684,334.224,-156.304,169.999,53.256,160.420
C03241=1009.679,333.976,-156.270,169.991,53.262,160.420
C03242=1009.673,333.729,-156.236,169.984,53.266,160.419
C03243=1009.666,333.481,-156.202,169.977,53.272,160.419
C03244=1009.660,333.233,-156.168,169.969,53.277,160.419
C03245=1009.654,332.986,-156.134,169.961,53.282,160.418
C03246=1009.648,332.737,-156.100,169.953,53.288,160.418
C03247=1009.642,332.490,-156.066,169.946,53.293,160.418
C03248=1009.637,332.243,-156.032,169.938,53.298,160.417
C03249=1009.630,331.995,-155.999,169.930,53.304,160.417
C03250=1009.624,331.747,-155.965,169.922,53.309,160.417
C03251=1009.618,331.500,-155.931,169.915,53.315,160.416
C03252=1009.612,331.252,-155.897,169.908,53.319,160.416
C03253=1009.607,331.005,-155.863,169.900,53.325,160.416
C03254=1009.600,330.756,-155.830,169.892,53.330,160.415
C03255=1009.594,330.509,-155.796,169.885,53.336,160.415
C03256=1009.588,330.261,-155.763,169.877,53.342,160.415
C03257=1009.582,330.014,-155.729,169.869,53.347,160.415
C03258=1009.576,329.766,-155.696,169.861,53.352,160.414
C03259=1009.569,329.518,-155.663,169.854,53.358,160.414
C03260=1009.563,329.271,-155.629,169.846,53.363,160.413
C03261=1009.558,329.023,-155.596,169.838,53.369,160.413
C03262=1009.551,328.775,-155.563,169.832,53.374,160.413
C03263=1009.546,328.528,-155.529,169.824,53.379,160.413
C03264=1009.540,328.280,-155.495,169.816,53.385,160.412
C03265=1009.534,328.033,-155.463,169.809,53.391,160.412
C03266=1009.528,327.785,-155.429,169.801,53.396,160.412
C03267=1009.523,327.537,-155.396,169.793,53.402,160.412
C03268=1009.516,327.290,-155.363,169.786,53.407,160.411
C03269=1009.511,327.042,-155.329,169.779,53.412,160.411
C03270=1009.504,326.794,-155.296,169.772,53.418,160.411
C03271=1009.499,326.546,-155.263,169.764,53.424,160.411
C03272=1009.493,326.298,-155.230,169.757,53.430,160.410
C03273=1009.487,326.051,-155.197,169.749,53.435,160.410
C03274=1009.481,325.803,-155.164,169.741,53.441,160.410
C03275=1009.476,325.555,-155.130,169.734,53.447,160.410
C03276=1009.469,325.308,-155.098,169.727,53.452,160.409
C03277=1009.464,325.060,-155.064,169.720,53.457,160.409
C03278=1009.458,324.812,-155.032,169.712,53.464,160.409
C03279=1009.451,324.564,-154.999,169.705,53.469,160.409
C03280=1009.444,324.232,-154.955,169.694,53.477,160.408
C03281=1009.435,323.899,-154.912,169.685,53.485,160.408
C03282=1009.427,323.567,-154.868,169.675,53.492,160.408
C03283=1009.419,323.234,-154.824,169.665,53.500,160.408
C03284=1009.413,322.987,-154.792,169.658,53.505,160.407
C03285=1009.408,322.739,-154.759,169.651,53.511,160.407
C03286=1009.402,322.491,-154.727,169.643,53.517,160.407
C03287=1009.396,322.244,-154.694,169.636,53.523,160.407
C03288=1009.390,321.995,-154.662,169.629,53.529,160.407
C03289=1009.383,321.748,-154.629,169.621,53.535,160.406
C03290=1009.378,321.500,-154.597,169.614,53.541,160.406
C03291=1009.372,321.252,-154.564,169.607,53.546,160.406
C03292=1009.366,321.004,-154.532,169.600,53.552,160.406
C03293=1009.360,320.756,-154.500,169.592,53.558,160.406
C03294=1009.355,320.509,-154.468,169.585,53.563,160.406
C03295=1009.349,320.261,-154.436,169.578,53.570,160.405
C03296=1009.342,320.013,-154.403,169.571,53.575,160.405
C03297=1009.338,319.765,-154.371,169.564,53.581,160.405
C03298=1009.332,319.517,-154.339,169.557,53.587,160.405
C03299=1009.326,319.270,-154.306,169.549,53.593,160.405
C03300=1009.320,319.022,-154.274,169.542,53.599,160.405
C03301=1009.314,318.774,-154.242,169.534,53.605,160.404
C03302=1009.309,318.525,-154.210,169.528,53.611,160.404
C03303=1009.303,318.278,-154.177,169.521,53.617,160.404
C03304=1009.297,318.030,-154.145,169.513,53.623,160.404
C03305=1009.292,317.783,-154.114,169.506,53.629,160.404
C03306=1009.286,317.535,-154.081,169.499,53.635,160.404
C03307=1009.280,317.288,-154.049,169.492,53.640,160.404
C03308=1009.275,317.039,-154.016,169.485,53.647,160.404
C03309=1009.269,316.791,-153.984,169.478,53.653,160.404
C03310=1009.264,316.543,-153.953,169.470,53.658,160.403
C03311=1009.258,316.295,-153.921,169.464,53.664,160.403
C03312=1009.252,316.048,-153.889,169.457,53.671,160.403
C03313=1009.247,315.800,-153.857,169.450,53.677,160.403
C03314=1009.242,315.552,-153.825,169.442,53.682,160.403
C03315=1009.236,315.304,-153.793,169.435,53.689,160.403
C03316=1009.230,315.056,-153.761,169.429,53.695,160.403
C03317=1009.225,314.808,-153.729,169.422,53.701,160.403
C03318=1009.219,314.560,-153.697,169.414,53.707,160.403
C03319=1009.213,314.313,-153.666,169.407,53.713,160.402
C03320=1009.209,314.065,-153.634,169.401,53.719,160.402
C03321=1009.203,313.817,-153.602,169.393,53.725,160.402
C03322=1009.197,313.569,-153.570,169.386,53.731,160.402
C03323=1009.192,313.322,-153.538,169.379,53.737,160.402
C03324=1009.186,313.073,-153.506,169.373,53.743,160.402
C03325=1009.181,312.825,-153.475,169.366,53.750,160.402
C03326=1009.176,312.577,-153.443,169.359,53.756,160.402
C03327=1009.171,312.330,-153.411,169.351,53.762,160.402
C03328=1009.165,312.082,-153.379,169.345,53.768,160.402
C03329=1009.160,311.834,-153.348,169.338,53.774,160.402
C03330=1009.154,311.586,-153.317,169.331,53.781,160.402
C03331=1009.149,311.339,-153.285,169.325,53.787,160.402
C03332=1009.144,311.090,-153.252,169.318,53.793,160.402
C03333=1009.139,310.842,-153.221,169.310,53.799,160.402
C03334=1009.133,310.594,-153.190,169.303,53.805,160.402
C03335=1009.128,310.347,-153.158,169.297,53.811,160.402
C03336=1009.123,310.099,-153.127,169.290,53.818,160.402
C03337=1009.117,309.851,-153.096,169.283,53.824,160.401
C03338=1009.112,309.603,-153.063,169.277,53.830,160.401
C03339=1009.107,309.355,-153.032,169.269,53.836,160.401
C03340=1009.100,309.028,-152.990,169.260,53.844,160.401
C03341=1009.093,308.701,-152.949,169.252,53.853,160.401
C03342=1009.087,308.375,-152.908,169.242,53.861,160.401
C03343=1009.079,308.048,-152.867,169.234,53.869,160.401
C03344=1009.073,307.800,-152.837,169.226,53.876,160.401
C03345=1009.068,307.552,-152.806,169.219,53.882,160.401
C03346=1009.063,307.305,-152.775,169.214,53.889,160.401
C03347=1009.057,307.056,-152.744,169.206,53.895,160.401
C03348=1009.051,306.808,-152.714,169.199,53.901,160.401
C03349=1009.046,306.560,-152.683,169.193,53.908,160.401
C03350=1009.040,306.312,-152.652,169.186,53.914,160.401
C03351=1009.035,306.064,-152.621,169.179,53.920,160.401
C03352=1009.029,305.816,-152.591,169.173,53.927,160.401
C03353=1009.024,305.568,-152.560,169.165,53.934,160.401
C03354=1009.018,305.320,-152.530,169.159,53.940,160.401
C03355=1009.013,305.072,-152.499,169.153,53.947,160.401
C03356=1009.007,304.824,-152.468,169.145,53.953,160.401
C03357=1009.002,304.576,-152.437,169.139,53.960,160.402
C03358=1008.997,304.328,-152.406,169.133,53.966,160.402
C03359=1008.991,304.080,-152.376,169.126,53.973,160.402
C03360=1008.986,303.832,-152.345,169.119,53.979,160.402
C03361=1008.981,303.584,-152.315,169.112,53.986,160.402
C03362=1008.976,303.335,-152.285,169.106,53.992,160.402
C03363=1008.971,303.088,-152.255,169.099,53.998,160.402
C03364=1008.965,302.840,-152.224,169.092,54.005,160.402
C03365=1008.960,302.592,-152.193,169.085,54.012,160.402
C03366=1008.955,302.343,-152.163,169.079,54.018,160.402
C03367=1008.949,302.096,-152.133,169.073,54.025,160.402
C03368=1008.944,301.847,-152.102,169.066,54.032,160.402
C03369=1008.938,301.600,-152.071,169.060,54.038,160.402
C03370=1008.934,301.352,-152.042,169.053,54.044,160.402
C03371=1008.928,301.104,-152.011,169.046,54.051,160.402
C03372=1008.923,300.856,-151.980,169.039,54.058,160.402
C03373=1008.918,300.607,-151.951,169.033,54.064,160.402
C03374=1008.913,300.359,-151.920,169.027,54.071,160.403
C03375=1008.908,300.111,-151.890,169.019,54.078,160.402
C03376=1008.903,299.863,-151.860,169.014,54.084,160.403
C03377=1008.897,299.615,-151.829,169.007,54.091,160.403
C03378=1008.892,299.367,-151.799,169.000,54.098,160.403
C03379=1008.887,299.120,-151.769,168.994,54.104,160.403
C03380=1008.883,298.893,-151.741,168.988,54.110,160.403
C03381=1008.878,298.667,-151.714,168.982,54.116,160.403
C03382=1008.873,298.442,-151.686,168.976,54.123,160.403
C03383=1008.868,298.215,-151.659,168.970,54.129,160.403
C03384=1008.864,297.989,-151.631,168.964,54.135,160.403
C03385=1008.860,297.763,-151.604,168.958,54.141,160.404
C03386=1008.854,297.538,-151.576,168.952,54.147,160.404
C03387=1008.850,297.312,-151.550,168.946,54.153,160.404
C03388=1008.609,298.138,-152.015,168.944,54.185,160.410
C03389=1008.614,298.391,-152.045,168.951,54.178,160.410
C03390=1008.620,298.644,-152.076,168.957,54.171,160.410
C03391=1008.624,298.897,-152.107,168.964,54.165,160.410
C03392=1008.629,299.149,-152.138,168.970,54.158,160.410
C03393=1008.634,299.398,-152.168,168.977,54.151,160.410
C03394=1008.640,299.646,-152.198,168.984,54.144,160.410
C03395=1008.645,299.894,-152.228,168.990,54.138,160.410
C03396=1008.650,300.142,-152.258,168.997,54.131,160.410
C03397=1008.655,300.390,-152.289,169.004,54.124,160.410
C03398=1008.660,300.638,-152.319,169.009,54.118,160.409
C03399=1008.665,300.886,-152.349,169.017,54.111,160.410
C03400=1008.670,301.134,-152.379,169.023,54.104,160.409
C03401=1008.676,301.382,-152.410,169.029,54.098,160.409
C03402=1008.681,301.631,-152.440,169.036,54.091,160.409
C03403=1008.686,301.879,-152.471,169.043,54.085,160.409
C03404=1008.691,302.126,-152.501,169.050,54.078,160.409
C03405=1008.696,302.375,-152.531,169.056,54.072,160.409
C03406=1008.702,302.622,-152.561,169.063,54.065,160.409
C03407=1008.707,302.871,-152.592,169.070,54.059,160.409
C03408=1008.713,303.119,-152.622,169.075,54.052,160.409
C03409=1008.718,303.367,-152.653,169.083,54.046,160.409
C03410=1008.723,303.615,-152.683,169.090,54.039,160.409
C03411=1008.728,303.862,-152.714,169.096,54.032,160.409
C03412=1008.734,304.110,-152.744,169.103,54.027,160.409
C03413=1008.738,304.359,-152.774,169.109,54.020,160.409
C03414=1008.744,304.607,-152.805,169.116,54.013,160.409
C03415=1008.749,304.855,-152.836,169.123,54.007,160.409
C03416=1008.755,305.103,-152.866,169.129,54.000,160.409
C03417=1008.760,305.351,-152.897,169.136,53.994,160.409
C03418=1008.766,305.599,-152.927,169.144,53.988,160.409
C03419=1008.771,305.847,-152.958,169.149,53.981,160.409
C03420=1008.776,306.095,-152.989,169.156,53.975,160.409
C03421=1008.782,306.343,-153.020,169.164,53.968,160.409
C03422=1008.787,306.591,-153.051,169.170,53.961,160.409
C03423=1008.793,306.839,-153.081,169.176,53.955,160.409
C03424=1008.798,307.087,-153.112,169.184,53.949,160.409
C03425=1008.804,307.335,-153.142,169.191,53.943,160.409
C03426=1008.809,307.583,-153.173,169.197,53.936,160.409
C03427=1008.815,307.831,-153.203,169.204,53.930,160.409
C03428=1008.820,308.079,-153.235,169.211,53.924,160.409
C03429=1008.828,308.408,-153.275,169.220,53.915,160.409
C03430=1008.834,308.737,-153.316,169.229,53.907,160.409
C03431=1008.841,309.066,-153.359,169.238,53.899,160.409
C03432=1008.848,309.395,-153.400,169.247,53.890,160.409
C03433=1008.853,309.643,-153.432,169.254,53.884,160.409
C03434=1008.859,309.891,-153.464,169.261,53.878,160.409
C03435=1008.864,310.139,-153.495,169.268,53.871,160.409
C03436=1008.869,310.386,-153.526,169.274,53.866,160.409
C03437=1008.874,310.635,-153.557,169.281,53.859,160.409
C03438=1008.879,310.882,-153.589,169.288,53.853,160.409
C03439=1008.885,311.131,-153.622,169.295,53.847,160.409
C03440=1008.890,311.379,-153.653,169.302,53.841,160.410
C03441=1008.895,311.626,-153.684,169.309,53.834,160.410
C03442=1008.901,311.874,-153.716,169.316,53.828,160.410
C03443=1008.906,312.122,-153.747,169.322,53.822,160.410
C03444=1008.912,312.370,-153.779,169.329,53.816,160.410
C03445=1008.916,312.618,-153.811,169.337,53.810,160.410
C03446=1008.922,312.865,-153.843,169.344,53.804,160.410
C03447=1008.927,313.114,-153.874,169.350,53.798,160.410
C03448=1008.933,313.362,-153.906,169.358,53.792,160.410
C03449=1008.938,313.609,-153.937,169.365,53.786,160.410
C03450=1008.943,313.857,-153.969,169.371,53.780,160.410
C03451=1008.949,314.105,-154.002,169.378,53.773,160.410
C03452=1008.954,314.353,-154.033,169.385,53.767,160.410
C03453=1008.959,314.600,-154.065,169.393,53.761,160.411
C03454=1008.965,314.849,-154.096,169.399,53.756,160.411
C03455=1008.971,315.097,-154.128,169.406,53.749,160.411
C03456=1008.976,315.344,-154.160,169.413,53.743,160.411
C03457=1008.981,315.593,-154.192,169.421,53.737,160.411
C03458=1008.987,315.840,-154.224,169.428,53.731,160.411
C03459=1008.993,316.088,-154.256,169.434,53.725,160.411
C03460=1008.998,316.336,-154.288,169.441,53.719,160.411
C03461=1009.003,316.583,-154.319,169.449,53.713,160.412
C03462=1009.009,316.832,-154.351,169.456,53.707,160.412
C03463=1009.014,317.079,-154.384,169.462,53.701,160.412
C03464=1009.020,317.327,-154.416,169.470,53.696,160.412
C03465=1009.026,317.575,-154.448,169.477,53.689,160.412
C03466=1009.032,317.823,-154.480,169.484,53.683,160.412
C03467=1009.038,318.071,-154.512,169.492,53.677,160.412
C03468=1009.043,318.319,-154.544,169.498,53.672,160.412
C03469=1009.048,318.567,-154.576,169.506,53.666,160.413
C03470=1009.054,318.814,-154.609,169.513,53.660,160.413
C03471=1009.060,319.062,-154.641,169.521,53.654,160.413
C03472=1009.065,319.310,-154.672,169.528,53.648,160.413
C03473=1009.071,319.558,-154.704,169.534,53.642,160.413
C03474=1009.078,319.805,-154.737,169.542,53.636,160.413
C03475=1009.082,320.053,-154.769,169.549,53.630,160.414
C03476=1009.088,320.302,-154.801,169.556,53.625,160.414
C03477=1009.095,320.549,-154.834,169.564,53.618,160.414
C03478=1009.100,320.797,-154.866,169.571,53.613,160.414
C03479=1009.106,321.045,-154.898,169.578,53.607,160.414
C03480=1009.112,321.292,-154.931,169.585,53.601,160.415
C03481=1009.117,321.540,-154.963,169.593,53.596,160.415
C03482=1009.123,321.788,-154.996,169.600,53.589,160.415
C03483=1009.129,322.036,-155.028,169.607,53.584,160.415
C03484=1009.135,322.284,-155.060,169.615,53.578,160.415
C03485=1009.141,322.532,-155.092,169.621,53.572,160.415
C03486=1009.146,322.779,-155.125,169.629,53.567,160.416
C03487=1009.152,323.027,-155.157,169.636,53.560,160.416
C03488=1009.159,323.275,-155.190,169.644,53.555,160.416
C03489=1009.167,323.609,-155.234,169.654,53.547,160.417
C03490=1009.174,323.945,-155.278,169.664,53.539,160.417
C03491=1009.183,324.280,-155.322,169.674,53.532,160.417
C03492=1009.191,324.614,-155.365,169.683,53.524,160.417
C03493=1009.197,324.862,-155.399,169.691,53.518,160.418
C03494=1009.202,325.109,-155.431,169.699,53.513,160.418
C03495=1009.208,325.357,-155.464,169.706,53.507,160.418
C03496=1009.214,325.604,-155.497,169.713,53.502,160.418
C03497=1009.220,325.852,-155.531,169.721,53.496,160.419
C03498=1009.226,326.100,-155.563,169.728,53.490,160.419
C03499=1009.232,326.348,-155.597,169.735,53.484,160.419
C03500=1009.237,326.596,-155.630,169.743,53.479,160.419
C03501=1009.244,326.843,-155.663,169.751,53.473,160.420
C03502=1009.249,327.091,-155.696,169.757,53.468,160.420
C03503=1009.255,327.339,-155.729,169.765,53.463,160.420
C03504=1009.261,327.587,-155.762,169.773,53.457,160.420
C03505=1009.267,327.835,-155.795,169.780,53.451,160.421
C03506=1009.273,328.082,-155.828,169.788,53.446,160.421
C03507=1009.279,328.330,-155.862,169.796,53.440,160.421
C03508=1009.284,328.577,-155.896,169.803,53.435,160.422
C03509=1009.291,328.825,-155.928,169.811,53.429,160.422
C03510=1009.296,329.073,-155.962,169.818,53.424,160.422
C03511=1009.302,329.320,-155.996,169.825,53.418,160.422
C03512=1009.308,329.568,-156.028,169.833,53.413,160.423
C03513=1009.314,329.816,-156.062,169.841,53.408,160.423
C03514=1009.320,330.064,-156.096,169.849,53.402,160.423
C03515=1009.327,330.311,-156.129,169.856,53.397,160.424
C03516=1009.332,330.559,-156.162,169.864,53.391,160.424
C03517=1009.339,330.806,-156.196,169.871,53.386,160.424
C03518=1009.344,331.054,-156.229,169.879,53.380,160.425
C03519=1009.351,331.302,-156.263,169.887,53.375,160.425
C03520=1009.356,331.550,-156.297,169.895,53.370,160.425
C03521=1009.363,331.797,-156.330,169.901,53.364,160.426
C03522=1009.368,332.045,-156.364,169.910,53.360,160.426
C03523=1009.374,332.292,-156.398,169.917,53.354,160.426
C03524=1009.381,332.540,-156.432,169.925,53.348,160.427
C03525=1009.386,332.788,-156.465,169.933,53.343,160.427
C03526=1009.392,333.035,-156.499,169.941,53.338,160.427
C03527=1009.399,333.283,-156.534,169.948,53.332,160.428
C03528=1009.404,333.531,-156.568,169.956,53.328,160.428
C03529=1009.410,333.778,-156.601,169.964,53.322,160.429
C03530=1009.417,334.026,-156.635,169.972,53.316,160.429
C03531=1009.423,334.273,-156.669,169.980,53.312,160.429
C03532=1009.429,334.521,-156.703,169.987,53.306,160.430
C03533=1009.435,334.769,-156.738,169.994,53.301,160.430
C03534=1009.441,335.016,-156.772,170.002,53.296,160.430
C03535=1009.447,335.265,-156.805,170.010,53.291,160.431
C03536=1009.453,335.512,-156.839,170.018,53.285,160.431
C03537=1009.459,335.759,-156.874,170.026,53.281,160.432
C03538=1009.466,336.007,-156.908,170.034,53.275,160.432
C03539=1009.472,336.254,-156.941,170.042,53.270,160.432
C03540=1009.479,336.502,-156.976,170.049,53.265,160.433
C03541=1009.485,336.749,-157.010,170.057,53.260,160.433
C03542=1009.491,336.997,-157.044,170.066,53.255,160.434
C03543=1009.497,337.245,-157.078,170.073,53.249,160.434
C03544=1009.503,337.493,-157.113,170.081,53.244,160.434
C03545=1009.509,337.739,-157.148,170.089,53.240,160.435
C03546=1009.516,337.987,-157.182,170.097,53.234,160.435
C03547=1009.522,338.235,-157.216,170.105,53.229,160.436
C03548=1009.528,338.483,-157.250,170.113,53.224,160.436
C03549=1009.537,338.813,-157.297,170.124,53.217,160.437
C03550=1009.545,339.143,-157.343,170.135,53.211,160.437
C03551=1009.553,339.473,-157.389,170.145,53.204,160.438
C03552=1009.561,339.803,-157.436,170.156,53.197,160.439
C03553=1009.568,340.051,-157.470,170.164,53.192,160.439
C03554=1009.575,340.299,-157.505,170.172,53.188,160.440
C03555=1009.580,340.546,-157.540,170.180,53.183,160.440
C03556=1009.587,340.793,-157.575,170.188,53.177,160.440
C03557=1009.593,341.042,-157.610,170.196,53.172,160.441
C03558=1009.600,341.289,-157.645,170.204,53.167,160.441
C03559=1009.606,341.536,-157.679,170.212,53.162,160.442
C03560=1009.612,341.784,-157.714,170.220,53.158,160.442
C03561=1009.619,342.031,-157.749,170.228,53.153,160.443
C03562=1009.625,342.279,-157.784,170.236,53.148,160.443
